ABB RobotStudio station: task2_Diaz_Raphael_20200421-193257.rsstn

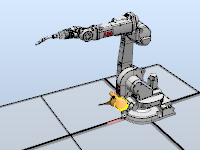
Station Solution2 (saved by RobotStudio 7.0.8732.594)
Controller IRB_1660ID_4kg_1.55m_1
  mechanical unit ROB_1: IRB1660ID_4_155__03, 6 joints, base frame (0, 0, 0) mm
Layout (positions relative to the parent item):
  - IRB1660ID_4_155__03 [mechanism, from Robots\IRB1660ID_4_155__03.rslib] at (0, 0, 0) mm; joint values [0, 0, 0, 0, 0, 0] (rad or m)
  - Binzel_ID_22 [mechanism, from Tools\Binzel_ID_22.rslib] at (962.96, 0, 1296.5) mm, rotated rx 0 ry 90 rz 0 deg
  - propeller [part, from Training Objects\propeller.rslib] at (600, 300, 492) mm
Attachment: Binzel_ID_22 is attached to IRB1660ID_4_155__03 / Link6
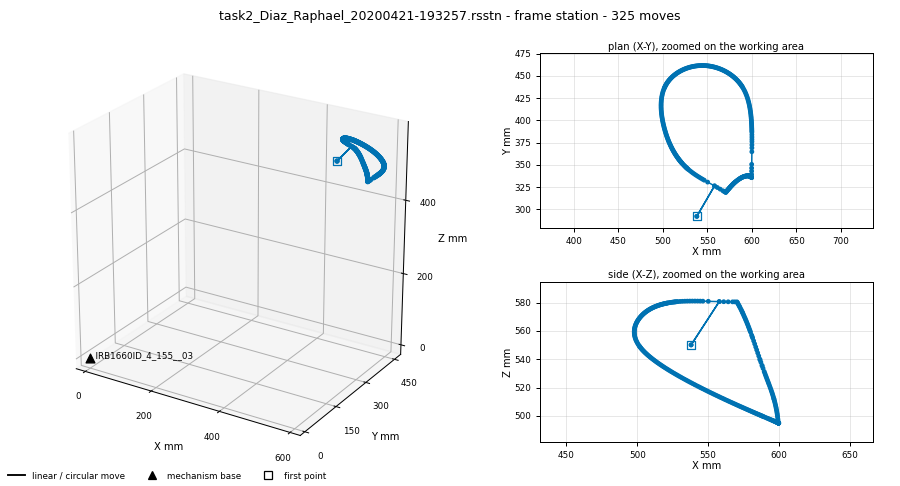
[picture p0: tool path of task2_Diaz_Raphael_20200421-193257.rsstn in frame station, 325 of 327 moves have a stored position in this frame; points joined in program order, loops and branches not executed]
Targets, tools, work objects and paths stored in the station, written as RAPID:
! task T_ROB1
MODULE CalibData
  PERS tooldata tWeldGun:=[TRUE,[[49.841566361,0,372.194826196],[0.981627183,0,0.190808995,0]],[2,[0,0,100],[0,1,0,0],0,0,0]];
  TASK PERS wobjdata wobjPropeller:=[FALSE,TRUE,"",[[600,300,492],[1,0,0,0]],[[0,0,0],[1,0,0,0]]];
ENDMODULE

! task T_ROB1
MODULE Module1
  CONST robtarget Target_10:=[[21.523963287,135.70517668,186.635026338],[0.089637387,-0.283764355,-0.851730307,0.431275333],[0,0,0,0],[9E+09,9E+09,9E+09,9E+09,9E+09,9E+09]];
  CONST robtarget Target_20:=[[-42.068819563,26.298976235,88.725674008],[0.089637387,-0.283764355,-0.851730307,0.431275333],[0,-1,-1,0],[9E+09,9E+09,9E+09,9E+09,9E+09,9E+09]];
  CONST robtarget Target_30:=[[-97.077163645,86.355573847,78.63839948],[0.089637387,-0.283764355,-0.851730307,0.431275333],[0,-1,-1,0],[9E+09,9E+09,9E+09,9E+09,9E+09,9E+09]];
  CONST robtarget Target_40:=[[-83.254485532,153.616685275,43.88735717],[0.089637387,-0.283764355,-0.851730307,0.431275333],[0,-1,-1,0],[9E+09,9E+09,9E+09,9E+09,9E+09,9E+09]];
  CONST robtarget Target_50:=[[-25.422721424,152.293184907,13.845629776],[0.089637387,-0.283764355,-0.851730307,0.431275333],[0,-1,-1,0],[9E+09,9E+09,9E+09,9E+09,9E+09,9E+09]];
  CONST robtarget Target_60:=[[-0.191127564,89.526890776,2.972180009],[0.089637387,-0.283764355,-0.851730307,0.431275333],[0,-1,-1,0],[9E+09,9E+09,9E+09,9E+09,9E+09,9E+09]];
  CONST robtarget Target_70:=[[-0.498093154,35.725710758,4.107130917],[0.089637387,-0.283764355,-0.851730307,0.431275333],[0,-1,-1,0],[9E+09,9E+09,9E+09,9E+09,9E+09,9E+09]];
  CONST robtarget Target_80:=[[-6.062970693,37.537743156,28.012491985],[0.089637387,-0.283764355,-0.851730307,0.431275333],[0,-1,-1,0],[9E+09,9E+09,9E+09,9E+09,9E+09,9E+09]];
  CONST robtarget Target_90:=[[-29.579108704,18.917792453,88.550574629],[0.089637387,-0.283764355,-0.851730307,0.431275333],[0,-1,-1,0],[9E+09,9E+09,9E+09,9E+09,9E+09,9E+09]];
  CONST robtarget Target_100:=[[-42.068819563,26.298976235,88.725674008],[0.089637387,-0.283764355,-0.851730307,0.431275333],[0,-1,-1,0],[9E+09,9E+09,9E+09,9E+09,9E+09,9E+09]];
  CONST robtarget Target_110:=[[-61.941679565,-7.890397172,58.129004558],[0.089637387,-0.283764355,-0.851730307,0.431275333],[0,-1,-1,0],[9E+09,9E+09,9E+09,9E+09,9E+09,9E+09]];
  CONST robtarget Target_120:=[[-61.941564206,-7.890461448,58.129001455],[0.089637387,-0.283764355,-0.851730307,0.431275333],[0,0,0,0],[9E+09,9E+09,9E+09,9E+09,9E+09,9E+09]];
  CONST robtarget Target_130:=[[-42.068819563,26.298976235,88.725674008],[0.089637387,-0.283764355,-0.851730307,0.431275333],[0,0,0,0],[9E+09,9E+09,9E+09,9E+09,9E+09,9E+09]];
  CONST robtarget Target_140:=[[-49.791866469,30.580230673,88.941782186],[0.089637387,-0.283764355,-0.851730307,0.431275333],[0,0,0,0],[9E+09,9E+09,9E+09,9E+09,9E+09,9E+09]];
  CONST robtarget Target_150:=[[-53.614959938,32.739613246,89.033496579],[0.089637387,-0.283764355,-0.851730307,0.431275333],[0,0,0,0],[9E+09,9E+09,9E+09,9E+09,9E+09,9E+09]];
  CONST robtarget Target_160:=[[-55.505547901,33.834166182,89.068675291],[0.089637387,-0.283764355,-0.851730307,0.431275333],[0,0,0,0],[9E+09,9E+09,9E+09,9E+09,9E+09,9E+09]];
  CONST robtarget Target_170:=[[-57.377839054,34.942502242,89.094223182],[0.089637387,-0.283764355,-0.851730307,0.431275333],[0,0,0,0],[9E+09,9E+09,9E+09,9E+09,9E+09,9E+09]];
  CONST robtarget Target_180:=[[-59.228590176,36.067527941,89.108256377],[0.089637387,-0.283764355,-0.851730307,0.431275333],[0,0,0,0],[9E+09,9E+09,9E+09,9E+09,9E+09,9E+09]];
  CONST robtarget Target_190:=[[-61.054558046,37.212149798,89.108891001],[0.089637387,-0.283764355,-0.851730307,0.431275333],[0,0,0,0],[9E+09,9E+09,9E+09,9E+09,9E+09,9E+09]];
  CONST robtarget Target_200:=[[-62.852499441,38.379274331,89.094243181],[0.089637387,-0.283764355,-0.851730307,0.431275333],[0,0,0,0],[9E+09,9E+09,9E+09,9E+09,9E+09,9E+09]];
  CONST robtarget Target_210:=[[-64.61917114,39.571808055,89.062429041],[0.089637387,-0.283764355,-0.851730307,0.431275333],[0,0,0,0],[9E+09,9E+09,9E+09,9E+09,9E+09,9E+09]];
  CONST robtarget Target_220:=[[-66.351329922,40.79265749,89.011564709],[0.089637387,-0.283764355,-0.851730307,0.431275333],[0,0,0,0],[9E+09,9E+09,9E+09,9E+09,9E+09,9E+09]];
  CONST robtarget Target_230:=[[-68.045732565,42.044729152,88.939766309],[0.089637387,-0.283764355,-0.851730307,0.431275333],[0,0,0,0],[9E+09,9E+09,9E+09,9E+09,9E+09,9E+09]];
  CONST robtarget Target_240:=[[-69.699135847,43.330929558,88.845149967],[0.089637387,-0.283764355,-0.851730307,0.431275333],[0,0,0,0],[9E+09,9E+09,9E+09,9E+09,9E+09,9E+09]];
  CONST robtarget Target_250:=[[-71.342075478,44.682787572,88.723134141],[0.089637387,-0.283764355,-0.851730307,0.431275333],[0,0,0,0],[9E+09,9E+09,9E+09,9E+09,9E+09,9E+09]];
  CONST robtarget Target_260:=[[-72.060749116,45.300688417,88.659667958],[0.089637387,-0.283764355,-0.851730307,0.431275333],[0,0,0,0],[9E+09,9E+09,9E+09,9E+09,9E+09,9E+09]];
  CONST robtarget Target_270:=[[-72.761042326,45.919421354,88.591393963],[0.089637387,-0.283764355,-0.851730307,0.431275333],[0,0,0,0],[9E+09,9E+09,9E+09,9E+09,9E+09,9E+09]];
  CONST robtarget Target_280:=[[-73.192658943,46.30937181,88.54602645],[0.089637387,-0.283764355,-0.851730307,0.431275333],[0,0,0,0],[9E+09,9E+09,9E+09,9E+09,9E+09,9E+09]];
  CONST robtarget Target_290:=[[-73.676857993,46.754481273,88.492204842],[0.089637387,-0.283764355,-0.851730307,0.431275333],[0,0,0,0],[9E+09,9E+09,9E+09,9E+09,9E+09,9E+09]];
  CONST robtarget Target_300:=[[-74.211820015,47.256226874,88.428916141],[0.089637387,-0.283764355,-0.851730307,0.431275333],[0,0,0,0],[9E+09,9E+09,9E+09,9E+09,9E+09,9E+09]];
  CONST robtarget Target_310:=[[-74.795612514,47.816163555,88.355085942],[0.089637387,-0.283764355,-0.851730307,0.431275333],[0,0,0,0],[9E+09,9E+09,9E+09,9E+09,9E+09,9E+09]];
  CONST robtarget Target_320:=[[-75.426303,48.435846257,88.269639843],[0.089637387,-0.283764355,-0.851730307,0.431275333],[0,0,0,0],[9E+09,9E+09,9E+09,9E+09,9E+09,9E+09]];
  CONST robtarget Target_330:=[[-76.101837442,49.116922118,88.171436479],[0.089637387,-0.283764355,-0.851730307,0.431275333],[0,0,0,0],[9E+09,9E+09,9E+09,9E+09,9E+09,9E+09]];
  CONST robtarget Target_340:=[[-76.819730038,49.861315108,88.059102158],[0.089637387,-0.283764355,-0.851730307,0.431275333],[0,0,0,0],[9E+09,9E+09,9E+09,9E+09,9E+09,9E+09]];
  CONST robtarget Target_350:=[[-77.577400632,50.670995418,87.931213982],[0.089637387,-0.283764355,-0.851730307,0.431275333],[0,0,0,0],[9E+09,9E+09,9E+09,9E+09,9E+09,9E+09]];
  CONST robtarget Target_360:=[[-78.37226907,51.547933238,87.786349051],[0.089637387,-0.283764355,-0.851730307,0.431275333],[0,0,0,0],[9E+09,9E+09,9E+09,9E+09,9E+09,9E+09]];
  CONST robtarget Target_370:=[[-78.78283064,52.012251515,87.70709705],[0.089637387,-0.283764355,-0.851730307,0.431275333],[0,0,0,0],[9E+09,9E+09,9E+09,9E+09,9E+09,9E+09]];
  CONST robtarget Target_380:=[[-79.201648961,52.494165078,87.623027502],[0.089637387,-0.283764355,-0.851730307,0.431275333],[0,0,0,0],[9E+09,9E+09,9E+09,9E+09,9E+09,9E+09]];
  CONST robtarget Target_390:=[[-79.628335409,52.993946989,87.533928686],[0.089637387,-0.283764355,-0.851730307,0.431275333],[0,0,0,0],[9E+09,9E+09,9E+09,9E+09,9E+09,9E+09]];
  CONST robtarget Target_400:=[[-80.062501358,53.511870309,87.439588878],[0.089637387,-0.283764355,-0.851730307,0.431275333],[0,0,0,0],[9E+09,9E+09,9E+09,9E+09,9E+09,9E+09]];
  CONST robtarget Target_410:=[[-80.503758184,54.048208097,87.339796355],[0.089637387,-0.283764355,-0.851730307,0.431275333],[0,0,0,0],[9E+09,9E+09,9E+09,9E+09,9E+09,9E+09]];
  CONST robtarget Target_420:=[[-80.951717264,54.603233414,87.234339393],[0.089637387,-0.283764355,-0.851730307,0.431275333],[0,0,0,0],[9E+09,9E+09,9E+09,9E+09,9E+09,9E+09]];
  CONST robtarget Target_430:=[[-81.405989972,55.177219322,87.123006269],[0.089637387,-0.283764355,-0.851730307,0.431275333],[0,0,0,0],[9E+09,9E+09,9E+09,9E+09,9E+09,9E+09]];
  CONST robtarget Target_440:=[[-81.866187684,55.77043888,87.005585259],[0.089637387,-0.283764355,-0.851730307,0.431275333],[0,0,0,0],[9E+09,9E+09,9E+09,9E+09,9E+09,9E+09]];
  CONST robtarget Target_450:=[[-82.331908288,56.383173791,86.881857385],[0.089637387,-0.283764355,-0.851730307,0.431275333],[0,0,0,0],[9E+09,9E+09,9E+09,9E+09,9E+09,9E+09]];
  CONST robtarget Target_460:=[[-82.802718317,57.015702111,86.751589396],[0.089637387,-0.283764355,-0.851730307,0.431275333],[0,0,0,0],[9E+09,9E+09,9E+09,9E+09,9E+09,9E+09]];
  CONST robtarget Target_470:=[[-83.278182117,57.668291429,86.614548166],[0.089637387,-0.283764355,-0.851730307,0.431275333],[0,0,0,0],[9E+09,9E+09,9E+09,9E+09,9E+09,9E+09]];
  CONST robtarget Target_480:=[[-83.75786403,58.341209334,86.470500568],[0.089637387,-0.283764355,-0.851730307,0.431275333],[0,0,0,0],[9E+09,9E+09,9E+09,9E+09,9E+09,9E+09]];
  CONST robtarget Target_490:=[[-84.2413284,59.034723416,86.319213476],[0.089637387,-0.283764355,-0.851730307,0.431275333],[0,0,0,0],[9E+09,9E+09,9E+09,9E+09,9E+09,9E+09]];
  CONST robtarget Target_500:=[[-84.728139572,59.749101264,86.160453763],[0.089637387,-0.283764355,-0.851730307,0.431275333],[0,0,0,0],[9E+09,9E+09,9E+09,9E+09,9E+09,9E+09]];
  CONST robtarget Target_510:=[[-85.21786189,60.484610466,85.993988302],[0.089637387,-0.283764355,-0.851730307,0.431275333],[0,0,0,0],[9E+09,9E+09,9E+09,9E+09,9E+09,9E+09]];
  CONST robtarget Target_520:=[[-85.710059697,61.241518614,85.819583966],[0.089637387,-0.283764355,-0.851730307,0.431275333],[0,0,0,0],[9E+09,9E+09,9E+09,9E+09,9E+09,9E+09]];
  CONST robtarget Target_530:=[[-86.204286606,62.020097275,85.637002174],[0.089637387,-0.283764355,-0.851730307,0.431275333],[0,0,0,0],[9E+09,9E+09,9E+09,9E+09,9E+09,9E+09]];
  CONST robtarget Target_540:=[[-86.700080407,62.820588107,85.446000215],[0.089637387,-0.283764355,-0.851730307,0.431275333],[0,0,0,0],[9E+09,9E+09,9E+09,9E+09,9E+09,9E+09]];
  CONST robtarget Target_550:=[[-87.196981704,63.643213831,85.246338775],[0.089637387,-0.283764355,-0.851730307,0.431275333],[0,0,0,0],[9E+09,9E+09,9E+09,9E+09,9E+09,9E+09]];
  CONST robtarget Target_560:=[[-87.694531106,64.488197169,85.037778537],[0.089637387,-0.283764355,-0.851730307,0.431275333],[0,0,0,0],[9E+09,9E+09,9E+09,9E+09,9E+09,9E+09]];
  CONST robtarget Target_570:=[[-88.192269217,65.355760842,84.820080186],[0.089637387,-0.283764355,-0.851730307,0.431275333],[0,0,0,0],[9E+09,9E+09,9E+09,9E+09,9E+09,9E+09]];
  CONST robtarget Target_580:=[[-88.689736644,66.246127572,84.593004406],[0.089637387,-0.283764355,-0.851730307,0.431275333],[0,0,0,0],[9E+09,9E+09,9E+09,9E+09,9E+09,9E+09]];
  CONST robtarget Target_590:=[[-89.186473995,67.159520081,84.356311882],[0.089637387,-0.283764355,-0.851730307,0.431275333],[0,0,0,0],[9E+09,9E+09,9E+09,9E+09,9E+09,9E+09]];
  CONST robtarget Target_600:=[[-89.682021875,68.09616109,84.109763297],[0.089637387,-0.283764355,-0.851730307,0.431275333],[0,0,0,0],[9E+09,9E+09,9E+09,9E+09,9E+09,9E+09]];
  CONST robtarget Target_610:=[[-90.175913619,69.056271448,83.853116141],[0.089637387,-0.283764355,-0.851730307,0.431275333],[0,0,0,0],[9E+09,9E+09,9E+09,9E+09,9E+09,9E+09]];
  CONST robtarget Target_620:=[[-90.667685083,70.040011068,83.586135756],[0.089637387,-0.283764355,-0.851730307,0.431275333],[0,0,0,0],[9E+09,9E+09,9E+09,9E+09,9E+09,9E+09]];
  CONST robtarget Target_630:=[[-91.15688065,71.04751127,83.308594608],[0.089637387,-0.283764355,-0.851730307,0.431275333],[0,0,0,0],[9E+09,9E+09,9E+09,9E+09,9E+09,9E+09]];
  CONST robtarget Target_640:=[[-91.643044702,72.078903372,83.020265165],[0.089637387,-0.283764355,-0.851730307,0.431275333],[0,0,0,0],[9E+09,9E+09,9E+09,9E+09,9E+09,9E+09]];
  CONST robtarget Target_650:=[[-92.125721625,73.134318692,82.720919892],[0.089637387,-0.283764355,-0.851730307,0.431275333],[0,0,0,0],[9E+09,9E+09,9E+09,9E+09,9E+09,9E+09]];
  CONST robtarget Target_660:=[[-92.604455801,74.21388855,82.410331256],[0.089637387,-0.283764355,-0.851730307,0.431275333],[0,0,0,0],[9E+09,9E+09,9E+09,9E+09,9E+09,9E+09]];
  CONST robtarget Target_670:=[[-93.078791613,75.317744264,82.088271723],[0.089637387,-0.283764355,-0.851730307,0.431275333],[0,0,0,0],[9E+09,9E+09,9E+09,9E+09,9E+09,9E+09]];
  CONST robtarget Target_680:=[[-93.548273446,76.446017152,81.754513761],[0.089637387,-0.283764355,-0.851730307,0.431275333],[0,0,0,0],[9E+09,9E+09,9E+09,9E+09,9E+09,9E+09]];
  CONST robtarget Target_690:=[[-94.012442576,77.598829619,81.408829359],[0.089637387,-0.283764355,-0.851730307,0.431275333],[0,0,0,0],[9E+09,9E+09,9E+09,9E+09,9E+09,9E+09]];
  CONST robtarget Target_700:=[[-94.470863955,78.776207351,81.051012179],[0.089637387,-0.283764355,-0.851730307,0.431275333],[0,0,0,0],[9E+09,9E+09,9E+09,9E+09,9E+09,9E+09]];
  CONST robtarget Target_710:=[[-94.92311748,79.978136589,80.6808672],[0.089637387,-0.283764355,-0.851730307,0.431275333],[0,0,0,0],[9E+09,9E+09,9E+09,9E+09,9E+09,9E+09]];
  CONST robtarget Target_720:=[[-95.368783045,81.204603576,80.298199397],[0.089637387,-0.283764355,-0.851730307,0.431275333],[0,0,0,0],[9E+09,9E+09,9E+09,9E+09,9E+09,9E+09]];
  CONST robtarget Target_730:=[[-95.807440548,82.455594554,79.902813746],[0.089637387,-0.283764355,-0.851730307,0.431275333],[0,0,0,0],[9E+09,9E+09,9E+09,9E+09,9E+09,9E+09]];
  CONST robtarget Target_740:=[[-96.238669885,83.731095764,79.494515226],[0.089637387,-0.283764355,-0.851730307,0.431275333],[0,0,0,0],[9E+09,9E+09,9E+09,9E+09,9E+09,9E+09]];
  CONST robtarget Target_750:=[[-96.662050952,85.031093447,79.073108811],[0.089637387,-0.283764355,-0.851730307,0.431275333],[0,0,0,0],[9E+09,9E+09,9E+09,9E+09,9E+09,9E+09]];
  CONST robtarget Target_760:=[[-97.077163645,86.355573847,78.63839948],[0.089637387,-0.283764355,-0.851730307,0.431275333],[0,0,0,0],[9E+09,9E+09,9E+09,9E+09,9E+09,9E+09]];
  CONST robtarget Target_770:=[[-97.483682077,87.704485468,78.19021474],[0.089637387,-0.283764355,-0.851730307,0.431275333],[0,0,0,0],[9E+09,9E+09,9E+09,9E+09,9E+09,9E+09]];
  CONST robtarget Target_780:=[[-97.881197354,89.077633701,77.728399267],[0.089637387,-0.283764355,-0.851730307,0.431275333],[0,0,0,0],[9E+09,9E+09,9E+09,9E+09,9E+09,9E+09]];
  CONST robtarget Target_790:=[[-98.269164855,90.47479012,77.252783791],[0.089637387,-0.283764355,-0.851730307,0.431275333],[0,0,0,0],[9E+09,9E+09,9E+09,9E+09,9E+09,9E+09]];
  CONST robtarget Target_800:=[[-98.647039962,91.895726298,76.763199041],[0.089637387,-0.283764355,-0.851730307,0.431275333],[0,0,0,0],[9E+09,9E+09,9E+09,9E+09,9E+09,9E+09]];
  CONST robtarget Target_810:=[[-99.013905738,93.340048971,76.259451373],[0.089637387,-0.283764355,-0.851730307,0.431275333],[0,0,0,0],[9E+09,9E+09,9E+09,9E+09,9E+09,9E+09]];
  CONST robtarget Target_820:=[[-99.368243888,94.807039694,75.741321273],[0.089637387,-0.283764355,-0.851730307,0.431275333],[0,0,0,0],[9E+09,9E+09,9E+09,9E+09,9E+09,9E+09]];
  CONST robtarget Target_830:=[[-99.708607753,96.295982268,75.208600662],[0.089637387,-0.283764355,-0.851730307,0.431275333],[0,0,0,0],[9E+09,9E+09,9E+09,9E+09,9E+09,9E+09]];
  CONST robtarget Target_840:=[[-100.033550677,97.806160497,74.661081462],[0.089637387,-0.283764355,-0.851730307,0.431275333],[0,0,0,0],[9E+09,9E+09,9E+09,9E+09,9E+09,9E+09]];
  CONST robtarget Target_850:=[[-100.341583594,99.336818217,74.098557633],[0.089637387,-0.283764355,-0.851730307,0.431275333],[0,0,0,0],[9E+09,9E+09,9E+09,9E+09,9E+09,9E+09]];
  CONST robtarget Target_860:=[[-100.631031883,100.8870215,73.520833315],[0.089637387,-0.283764355,-0.851730307,0.431275333],[0,0,0,0],[9E+09,9E+09,9E+09,9E+09,9E+09,9E+09]];
  CONST robtarget Target_870:=[[-100.900170557,102.455787493,72.927715696],[0.089637387,-0.283764355,-0.851730307,0.431275333],[0,0,0,0],[9E+09,9E+09,9E+09,9E+09,9E+09,9E+09]];
  CONST robtarget Target_880:=[[-101.147274629,104.042133343,72.319011966],[0.089637387,-0.283764355,-0.851730307,0.431275333],[0,0,0,0],[9E+09,9E+09,9E+09,9E+09,9E+09,9E+09]];
  CONST robtarget Target_890:=[[-101.370571802,105.645030719,71.694531974],[0.089637387,-0.283764355,-0.851730307,0.431275333],[0,0,0,0],[9E+09,9E+09,9E+09,9E+09,9E+09,9E+09]];
  CONST robtarget Target_900:=[[-101.568083835,107.263250566,71.054098336],[0.089637387,-0.283764355,-0.851730307,0.431275333],[0,0,0,0],[9E+09,9E+09,9E+09,9E+09,9E+09,9E+09]];
  CONST robtarget Target_910:=[[-101.737776824,108.895508939,70.397537389],[0.089637387,-0.283764355,-0.851730307,0.431275333],[0,0,0,0],[9E+09,9E+09,9E+09,9E+09,9E+09,9E+09]];
  CONST robtarget Target_920:=[[-101.877616866,110.540521898,69.724675469],[0.089637387,-0.283764355,-0.851730307,0.431275333],[0,0,0,0],[9E+09,9E+09,9E+09,9E+09,9E+09,9E+09]];
  CONST robtarget Target_930:=[[-101.985517598,112.196954226,69.035342228],[0.089637387,-0.283764355,-0.851730307,0.431275333],[0,0,0,0],[9E+09,9E+09,9E+09,9E+09,9E+09,9E+09]];
  CONST robtarget Target_940:=[[-102.059165334,113.863245906,68.329382794],[0.089637387,-0.283764355,-0.851730307,0.431275333],[0,0,0,0],[9E+09,9E+09,9E+09,9E+09,9E+09,9E+09]];
  CONST robtarget Target_950:=[[-102.096185174,115.537775795,67.606646723],[0.089637387,-0.283764355,-0.851730307,0.431275333],[0,0,0,0],[9E+09,9E+09,9E+09,9E+09,9E+09,9E+09]];
  CONST robtarget Target_960:=[[-102.094202223,117.218922746,66.866983568],[0.089637387,-0.283764355,-0.851730307,0.431275333],[0,0,0,0],[9E+09,9E+09,9E+09,9E+09,9E+09,9E+09]];
  CONST robtarget Target_970:=[[-102.050783732,118.905008267,66.110246882],[0.089637387,-0.283764355,-0.851730307,0.431275333],[0,0,0,0],[9E+09,9E+09,9E+09,9E+09,9E+09,9E+09]];
  CONST robtarget Target_980:=[[-101.963247246,120.594103871,65.336308536],[0.089637387,-0.283764355,-0.851730307,0.431275333],[0,0,0,0],[9E+09,9E+09,9E+09,9E+09,9E+09,9E+09]];
  CONST robtarget Target_990:=[[-101.82884331,122.284213421,64.545045559],[0.089637387,-0.283764355,-0.851730307,0.431275333],[0,0,0,0],[9E+09,9E+09,9E+09,9E+09,9E+09,9E+09]];
  CONST robtarget Target_1000:=[[-101.644822469,123.973340779,63.736334981],[0.089637387,-0.283764355,-0.851730307,0.431275333],[0,0,0,0],[9E+09,9E+09,9E+09,9E+09,9E+09,9E+09]];
  CONST robtarget Target_1010:=[[-101.408371772,125.659426107,62.910058546],[0.089637387,-0.283764355,-0.851730307,0.431275333],[0,0,0,0],[9E+09,9E+09,9E+09,9E+09,9E+09,9E+09]];
  CONST robtarget Target_1020:=[[-101.116405192,127.340133258,62.066119282],[0.089637387,-0.283764355,-0.851730307,0.431275333],[0,0,0,0],[9E+09,9E+09,9E+09,9E+09,9E+09,9E+09]];
  CONST robtarget Target_1030:=[[-100.765763661,129.013051638,61.204426141],[0.089637387,-0.283764355,-0.851730307,0.431275333],[0,0,0,0],[9E+09,9E+09,9E+09,9E+09,9E+09,9E+09]];
  CONST robtarget Target_1040:=[[-100.353288111,130.675770651,60.324888075],[0.089637387,-0.283764355,-0.851730307,0.431275333],[0,0,0,0],[9E+09,9E+09,9E+09,9E+09,9E+09,9E+09]];
  CONST robtarget Target_1050:=[[-99.875750085,132.325809364,59.4274195],[0.089637387,-0.283764355,-0.851730307,0.431275333],[0,0,0,0],[9E+09,9E+09,9E+09,9E+09,9E+09,9E+09]];
  CONST robtarget Target_1060:=[[-99.329623689,133.96038311,58.511959204],[0.089637387,-0.283764355,-0.851730307,0.431275333],[0,0,0,0],[9E+09,9E+09,9E+09,9E+09,9E+09,9E+09]];
  CONST robtarget Target_1070:=[[-98.711303696,135.57662569,57.578452699],[0.089637387,-0.283764355,-0.851730307,0.431275333],[0,0,0,0],[9E+09,9E+09,9E+09,9E+09,9E+09,9E+09]];
  CONST robtarget Target_1080:=[[-98.373944468,136.376977106,57.10491509],[0.089637387,-0.283764355,-0.851730307,0.431275333],[0,0,0,0],[9E+09,9E+09,9E+09,9E+09,9E+09,9E+09]];
  CONST robtarget Target_1090:=[[-98.01718488,137.171670907,56.626845496],[0.089637387,-0.283764355,-0.851730307,0.431275333],[0,0,0,0],[9E+09,9E+09,9E+09,9E+09,9E+09,9E+09]];
  CONST robtarget Target_1100:=[[-97.640535504,137.960322993,56.144237301],[0.089637387,-0.283764355,-0.851730307,0.431275333],[0,0,0,0],[9E+09,9E+09,9E+09,9E+09,9E+09,9E+09]];
  CONST robtarget Target_1110:=[[-97.243501368,138.742523396,55.657088796],[0.089637387,-0.283764355,-0.851730307,0.431275333],[0,0,0,0],[9E+09,9E+09,9E+09,9E+09,9E+09,9E+09]];
  CONST robtarget Target_1120:=[[-96.825623509,139.517875036,55.165400527],[0.089637387,-0.283764355,-0.851730307,0.431275333],[0,0,0,0],[9E+09,9E+09,9E+09,9E+09,9E+09,9E+09]];
  CONST robtarget Target_1130:=[[-96.386442962,140.28598083,54.669173042],[0.089637387,-0.283764355,-0.851730307,0.431275333],[0,0,0,0],[9E+09,9E+09,9E+09,9E+09,9E+09,9E+09]];
  CONST robtarget Target_1140:=[[-95.925711374,141.046481587,54.168428273],[0.089637387,-0.283764355,-0.851730307,0.431275333],[0,0,0,0],[9E+09,9E+09,9E+09,9E+09,9E+09,9E+09]];
  CONST robtarget Target_1150:=[[-95.443552762,141.799075074,53.663228181],[0.089637387,-0.283764355,-0.851730307,0.431275333],[0,0,0,0],[9E+09,9E+09,9E+09,9E+09,9E+09,9E+09]];
  CONST robtarget Target_1160:=[[-94.940066713,142.543449653,53.153633355],[0.089637387,-0.283764355,-0.851730307,0.431275333],[0,0,0,0],[9E+09,9E+09,9E+09,9E+09,9E+09,9E+09]];
  CONST robtarget Target_1170:=[[-94.415352815,143.279293685,52.639704389],[0.089637387,-0.283764355,-0.851730307,0.431275333],[0,0,0,0],[9E+09,9E+09,9E+09,9E+09,9E+09,9E+09]];
  CONST robtarget Target_1180:=[[-93.869500391,144.006300939,52.121499208],[0.089637387,-0.283764355,-0.851730307,0.431275333],[0,0,0,0],[9E+09,9E+09,9E+09,9E+09,9E+09,9E+09]];
  CONST robtarget Target_1190:=[[-93.302636325,144.724144959,51.59908555],[0.089637387,-0.283764355,-0.851730307,0.431275333],[0,0,0,0],[9E+09,9E+09,9E+09,9E+09,9E+09,9E+09]];
  CONST robtarget Target_1200:=[[-92.71491655,145.432483766,51.072538723],[0.089637387,-0.283764355,-0.851730307,0.431275333],[0,0,0,0],[9E+09,9E+09,9E+09,9E+09,9E+09,9E+09]];
  CONST robtarget Target_1210:=[[-92.106496997,146.13097538,50.541934035],[0.089637387,-0.283764355,-0.851730307,0.431275333],[0,0,0,0],[9E+09,9E+09,9E+09,9E+09,9E+09,9E+09]];
  CONST robtarget Target_1220:=[[-91.477533598,146.819277823,50.007346793],[0.089637387,-0.283764355,-0.851730307,0.431275333],[0,0,0,0],[9E+09,9E+09,9E+09,9E+09,9E+09,9E+09]];
  CONST robtarget Target_1230:=[[-90.828182284,147.497049114,49.468852306],[0.089637387,-0.283764355,-0.851730307,0.431275333],[0,0,0,0],[9E+09,9E+09,9E+09,9E+09,9E+09,9E+09]];
  CONST robtarget Target_1240:=[[-90.158598987,148.163947276,48.926525883],[0.089637387,-0.283764355,-0.851730307,0.431275333],[0,0,0,0],[9E+09,9E+09,9E+09,9E+09,9E+09,9E+09]];
  CONST robtarget Target_1250:=[[-89.468939638,148.819630327,48.38044283],[0.089637387,-0.283764355,-0.851730307,0.431275333],[0,0,0,0],[9E+09,9E+09,9E+09,9E+09,9E+09,9E+09]];
  CONST robtarget Target_1260:=[[-88.759371673,149.463749958,47.83068148],[0.089637387,-0.283764355,-0.851730307,0.431275333],[0,0,0,0],[9E+09,9E+09,9E+09,9E+09,9E+09,9E+09]];
  CONST robtarget Target_1270:=[[-88.030117086,150.095929082,47.277334333],[0.089637387,-0.283764355,-0.851730307,0.431275333],[0,0,0,0],[9E+09,9E+09,9E+09,9E+09,9E+09,9E+09]];
  CONST robtarget Target_1280:=[[-87.281413645,150.715782558,46.72049795],[0.089637387,-0.283764355,-0.851730307,0.431275333],[0,0,0,0],[9E+09,9E+09,9E+09,9E+09,9E+09,9E+09]];
  CONST robtarget Target_1290:=[[-86.513499118,151.322925246,46.160268893],[0.089637387,-0.283764355,-0.851730307,0.431275333],[0,0,0,0],[9E+09,9E+09,9E+09,9E+09,9E+09,9E+09]];
  CONST robtarget Target_1300:=[[-85.726611275,151.916972002,45.596743725],[0.089637387,-0.283764355,-0.851730307,0.431275333],[0,0,0,0],[9E+09,9E+09,9E+09,9E+09,9E+09,9E+09]];
  CONST robtarget Target_1310:=[[-84.920987884,152.497537687,45.030019008],[0.089637387,-0.283764355,-0.851730307,0.431275333],[0,0,0,0],[9E+09,9E+09,9E+09,9E+09,9E+09,9E+09]];
  CONST robtarget Target_1320:=[[-84.096866713,153.064237158,44.460191302],[0.089637387,-0.283764355,-0.851730307,0.431275333],[0,0,0,0],[9E+09,9E+09,9E+09,9E+09,9E+09,9E+09]];
  CONST robtarget Target_1330:=[[-83.254485532,153.616685275,43.88735717],[0.089637387,-0.283764355,-0.851730307,0.431275333],[0,0,0,0],[9E+09,9E+09,9E+09,9E+09,9E+09,9E+09]];
  CONST robtarget Target_1340:=[[-82.394094894,154.154490046,43.311616509],[0.089637387,-0.283764355,-0.851730307,0.431275333],[0,0,0,0],[9E+09,9E+09,9E+09,9E+09,9E+09,9E+09]];
  CONST robtarget Target_1350:=[[-81.516005347,154.677228513,42.733084706],[0.089637387,-0.283764355,-0.851730307,0.431275333],[0,0,0,0],[9E+09,9E+09,9E+09,9E+09,9E+09,9E+09]];
  CONST robtarget Target_1360:=[[-80.620544648,155.184469083,42.151881558],[0.089637387,-0.283764355,-0.851730307,0.431275333],[0,0,0,0],[9E+09,9E+09,9E+09,9E+09,9E+09,9E+09]];
  CONST robtarget Target_1370:=[[-79.708040553,155.675780162,41.568126862],[0.089637387,-0.283764355,-0.851730307,0.431275333],[0,0,0,0],[9E+09,9E+09,9E+09,9E+09,9E+09,9E+09]];
  CONST robtarget Target_1380:=[[-78.778820818,156.150730158,40.981940416],[0.089637387,-0.283764355,-0.851730307,0.431275333],[0,0,0,0],[9E+09,9E+09,9E+09,9E+09,9E+09,9E+09]];
  CONST robtarget Target_1390:=[[-77.833213201,156.608887477,40.393442017],[0.089637387,-0.283764355,-0.851730307,0.431275333],[0,0,0,0],[9E+09,9E+09,9E+09,9E+09,9E+09,9E+09]];
  CONST robtarget Target_1400:=[[-76.871545457,157.049820527,39.802751462],[0.089637387,-0.283764355,-0.851730307,0.431275333],[0,0,0,0],[9E+09,9E+09,9E+09,9E+09,9E+09,9E+09]];
  CONST robtarget Target_1410:=[[-75.894145343,157.473097712,39.209988548],[0.089637387,-0.283764355,-0.851730307,0.431275333],[0,0,0,0],[9E+09,9E+09,9E+09,9E+09,9E+09,9E+09]];
  CONST robtarget Target_1420:=[[-74.901354733,157.878280056,38.615276732],[0.089637387,-0.283764355,-0.851730307,0.431275333],[0,0,0,0],[9E+09,9E+09,9E+09,9E+09,9E+09,9E+09]];
  CONST robtarget Target_1430:=[[-73.893581114,158.264895339,38.018756325],[0.089637387,-0.283764355,-0.851730307,0.431275333],[0,0,0,0],[9E+09,9E+09,9E+09,9E+09,9E+09,9E+09]];
  CONST robtarget Target_1440:=[[-72.87125067,158.632462113,37.420572413],[0.089637387,-0.283764355,-0.851730307,0.431275333],[0,0,0,0],[9E+09,9E+09,9E+09,9E+09,9E+09,9E+09]];
  CONST robtarget Target_1450:=[[-71.834789579,158.980498927,36.820870078],[0.089637387,-0.283764355,-0.851730307,0.431275333],[0,0,0,0],[9E+09,9E+09,9E+09,9E+09,9E+09,9E+09]];
  CONST robtarget Target_1460:=[[-70.784624025,159.308524331,36.219794405],[0.089637387,-0.283764355,-0.851730307,0.431275333],[0,0,0,0],[9E+09,9E+09,9E+09,9E+09,9E+09,9E+09]];
  CONST robtarget Target_1470:=[[-69.721180188,159.616056875,35.617490477],[0.089637387,-0.283764355,-0.851730307,0.431275333],[0,0,0,0],[9E+09,9E+09,9E+09,9E+09,9E+09,9E+09]];
  CONST robtarget Target_1480:=[[-68.644884249,159.902615109,35.014103378],[0.089637387,-0.283764355,-0.851730307,0.431275333],[0,0,0,0],[9E+09,9E+09,9E+09,9E+09,9E+09,9E+09]];
  CONST robtarget Target_1490:=[[-67.55616239,160.167717582,34.409778192],[0.089637387,-0.283764355,-0.851730307,0.431275333],[0,0,0,0],[9E+09,9E+09,9E+09,9E+09,9E+09,9E+09]];
  CONST robtarget Target_1500:=[[-66.455479479,160.410863431,33.804669917],[0.089637387,-0.283764355,-0.851730307,0.431275333],[0,0,0,0],[9E+09,9E+09,9E+09,9E+09,9E+09,9E+09]];
  CONST robtarget Target_1510:=[[-65.343353291,160.631525372,33.198947094],[0.089637387,-0.283764355,-0.851730307,0.431275333],[0,0,0,0],[9E+09,9E+09,9E+09,9E+09,9E+09,9E+09]];
  CONST robtarget Target_1520:=[[-64.220289368,160.829182326,32.592775118],[0.089637387,-0.283764355,-0.851730307,0.431275333],[0,0,0,0],[9E+09,9E+09,9E+09,9E+09,9E+09,9E+09]];
  CONST robtarget Target_1530:=[[-63.086793249,161.003313214,31.986319384],[0.089637387,-0.283764355,-0.851730307,0.431275333],[0,0,0,0],[9E+09,9E+09,9E+09,9E+09,9E+09,9E+09]];
  CONST robtarget Target_1540:=[[-61.943384215,161.153390145,31.379748799],[0.089637387,-0.283764355,-0.851730307,0.431275333],[0,0,0,0],[9E+09,9E+09,9E+09,9E+09,9E+09,9E+09]];
  CONST robtarget Target_1550:=[[-60.790609276,161.278871503,30.77323935],[0.089637387,-0.283764355,-0.851730307,0.431275333],[0,0,0,0],[9E+09,9E+09,9E+09,9E+09,9E+09,9E+09]];
  CONST robtarget Target_1560:=[[-59.629020895,161.379212994,30.166968412],[0.089637387,-0.283764355,-0.851730307,0.431275333],[0,0,0,0],[9E+09,9E+09,9E+09,9E+09,9E+09,9E+09]];
  CONST robtarget Target_1570:=[[-58.605848224,161.44595514,29.636819659],[0.089637387,-0.283764355,-0.851730307,0.431275333],[0,0,0,0],[9E+09,9E+09,9E+09,9E+09,9E+09,9E+09]];
  CONST robtarget Target_1580:=[[-57.318566058,161.500963653,28.974738132],[0.089637387,-0.283764355,-0.851730307,0.431275333],[0,0,0,0],[9E+09,9E+09,9E+09,9E+09,9E+09,9E+09]];
  CONST robtarget Target_1590:=[[-56.179983218,161.522654054,28.393499156],[0.089637387,-0.283764355,-0.851730307,0.431275333],[0,0,0,0],[9E+09,9E+09,9E+09,9E+09,9E+09,9E+09]];
  CONST robtarget Target_1600:=[[-55.043993927,161.519276456,27.817513287],[0.089637387,-0.283764355,-0.851730307,0.431275333],[0,0,0,0],[9E+09,9E+09,9E+09,9E+09,9E+09,9E+09]];
  CONST robtarget Target_1610:=[[-53.911152598,161.491173917,27.246893168],[0.089637387,-0.283764355,-0.851730307,0.431275333],[0,0,0,0],[9E+09,9E+09,9E+09,9E+09,9E+09,9E+09]];
  CONST robtarget Target_1620:=[[-52.782013645,161.438689493,26.681751443],[0.089637387,-0.283764355,-0.851730307,0.431275333],[0,0,0,0],[9E+09,9E+09,9E+09,9E+09,9E+09,9E+09]];
  CONST robtarget Target_1630:=[[-51.657131483,161.362166244,26.122200755],[0.089637387,-0.283764355,-0.851730307,0.431275333],[0,0,0,0],[9E+09,9E+09,9E+09,9E+09,9E+09,9E+09]];
  CONST robtarget Target_1640:=[[-50.537060524,161.261947226,25.568353747],[0.089637387,-0.283764355,-0.851730307,0.431275333],[0,0,0,0],[9E+09,9E+09,9E+09,9E+09,9E+09,9E+09]];
  CONST robtarget Target_1650:=[[-49.422355184,161.138375497,25.020323063],[0.089637387,-0.283764355,-0.851730307,0.431275333],[0,0,0,0],[9E+09,9E+09,9E+09,9E+09,9E+09,9E+09]];
  CONST robtarget Target_1660:=[[-48.31354999,160.991943178,24.478225714],[0.089637387,-0.283764355,-0.851730307,0.431275333],[0,0,0,0],[9E+09,9E+09,9E+09,9E+09,9E+09,9E+09]];
  CONST robtarget Target_1670:=[[-47.211113798,160.82319606,23.942165647],[0.089637387,-0.283764355,-0.851730307,0.431275333],[0,0,0,0],[9E+09,9E+09,9E+09,9E+09,9E+09,9E+09]];
  CONST robtarget Target_1680:=[[-46.115502514,160.632557701,23.412235913],[0.089637387,-0.283764355,-0.851730307,0.431275333],[0,0,0,0],[9E+09,9E+09,9E+09,9E+09,9E+09,9E+09]];
  CONST robtarget Target_1690:=[[-45.027172042,160.42045166,22.888529564],[0.089637387,-0.283764355,-0.851730307,0.431275333],[0,0,0,0],[9E+09,9E+09,9E+09,9E+09,9E+09,9E+09]];
  CONST robtarget Target_1700:=[[-43.946578289,160.187301498,22.371139651],[0.089637387,-0.283764355,-0.851730307,0.431275333],[0,0,0,0],[9E+09,9E+09,9E+09,9E+09,9E+09,9E+09]];
  CONST robtarget Target_1710:=[[-42.87417716,159.933530773,21.860159223],[0.089637387,-0.283764355,-0.851730307,0.431275333],[0,0,0,0],[9E+09,9E+09,9E+09,9E+09,9E+09,9E+09]];
  CONST robtarget Target_1720:=[[-41.810424561,159.659563045,21.355681333],[0.089637387,-0.283764355,-0.851730307,0.431275333],[0,0,0,0],[9E+09,9E+09,9E+09,9E+09,9E+09,9E+09]];
  CONST robtarget Target_1730:=[[-40.755776397,159.365821874,20.857799032],[0.089637387,-0.283764355,-0.851730307,0.431275333],[0,0,0,0],[9E+09,9E+09,9E+09,9E+09,9E+09,9E+09]];
  CONST robtarget Target_1740:=[[-39.710671647,159.052723834,20.366600679],[0.089637387,-0.283764355,-0.851730307,0.431275333],[0,0,0,0],[9E+09,9E+09,9E+09,9E+09,9E+09,9E+09]];
  CONST robtarget Target_1750:=[[-38.675489479,158.720660141,19.88215816],[0.089637387,-0.283764355,-0.851730307,0.431275333],[0,0,0,0],[9E+09,9E+09,9E+09,9E+09,9E+09,9E+09]];
  CONST robtarget Target_1760:=[[-37.650596085,158.370016319,19.404539813],[0.089637387,-0.283764355,-0.851730307,0.431275333],[0,0,0,0],[9E+09,9E+09,9E+09,9E+09,9E+09,9E+09]];
  CONST robtarget Target_1770:=[[-36.636357657,158.001177889,18.933813973],[0.089637387,-0.283764355,-0.851730307,0.431275333],[0,0,0,0],[9E+09,9E+09,9E+09,9E+09,9E+09,9E+09]];
  CONST robtarget Target_1780:=[[-35.633140386,157.614530375,18.470048979],[0.089637387,-0.283764355,-0.851730307,0.431275333],[0,0,0,0],[9E+09,9E+09,9E+09,9E+09,9E+09,9E+09]];
  CONST robtarget Target_1790:=[[-34.641310463,157.210459298,18.013313167],[0.089637387,-0.283764355,-0.851730307,0.431275333],[0,0,0,0],[9E+09,9E+09,9E+09,9E+09,9E+09,9E+09]];
  CONST robtarget Target_1800:=[[-33.661234081,156.789350181,17.563674874],[0.089637387,-0.283764355,-0.851730307,0.431275333],[0,0,0,0],[9E+09,9E+09,9E+09,9E+09,9E+09,9E+09]];
  CONST robtarget Target_1810:=[[-32.69327743,156.351588547,17.121202438],[0.089637387,-0.283764355,-0.851730307,0.431275333],[0,0,0,0],[9E+09,9E+09,9E+09,9E+09,9E+09,9E+09]];
  CONST robtarget Target_1820:=[[-31.737791053,155.897553351,16.685959875],[0.089637387,-0.283764355,-0.851730307,0.431275333],[0,0,0,0],[9E+09,9E+09,9E+09,9E+09,9E+09,9E+09]];
  CONST robtarget Target_1830:=[[-30.795070542,155.427599777,16.257996131],[0.089637387,-0.283764355,-0.851730307,0.431275333],[0,0,0,0],[9E+09,9E+09,9E+09,9E+09,9E+09,9E+09]];
  CONST robtarget Target_1840:=[[-29.865399659,154.942077691,15.837356936],[0.089637387,-0.283764355,-0.851730307,0.431275333],[0,0,0,0],[9E+09,9E+09,9E+09,9E+09,9E+09,9E+09]];
  CONST robtarget Target_1850:=[[-28.949062169,154.44133696,15.424088021],[0.089637387,-0.283764355,-0.851730307,0.431275333],[0,0,0,0],[9E+09,9E+09,9E+09,9E+09,9E+09,9E+09]];
  CONST robtarget Target_1860:=[[-28.046341837,153.92572745,15.018235117],[0.089637387,-0.283764355,-0.851730307,0.431275333],[0,0,0,0],[9E+09,9E+09,9E+09,9E+09,9E+09,9E+09]];
  CONST robtarget Target_1870:=[[-27.157522426,153.395599027,14.619843954],[0.089637387,-0.283764355,-0.851730307,0.431275333],[0,0,0,0],[9E+09,9E+09,9E+09,9E+09,9E+09,9E+09]];
  CONST robtarget Target_1880:=[[-26.2828877,152.851301557,14.228960264],[0.089637387,-0.283764355,-0.851730307,0.431275333],[0,0,0,0],[9E+09,9E+09,9E+09,9E+09,9E+09,9E+09]];
  CONST robtarget Target_1890:=[[-25.422721424,152.293184907,13.845629776],[0.089637387,-0.283764355,-0.851730307,0.431275333],[0,0,0,0],[9E+09,9E+09,9E+09,9E+09,9E+09,9E+09]];
  CONST robtarget Target_1900:=[[-24.577292951,151.721592779,13.469894259],[0.089637387,-0.283764355,-0.851730307,0.431275333],[0,0,0,0],[9E+09,9E+09,9E+09,9E+09,9E+09,9E+09]];
  CONST robtarget Target_1910:=[[-23.746821381,151.136846643,13.101781769],[0.089637387,-0.283764355,-0.851730307,0.431275333],[0,0,0,0],[9E+09,9E+09,9E+09,9E+09,9E+09,9E+09]];
  CONST robtarget Target_1920:=[[-22.931515099,150.539263009,12.741317469],[0.089637387,-0.283764355,-0.851730307,0.431275333],[0,0,0,0],[9E+09,9E+09,9E+09,9E+09,9E+09,9E+09]];
  CONST robtarget Target_1930:=[[-22.131582488,149.929158392,12.388526521],[0.089637387,-0.283764355,-0.851730307,0.431275333],[0,0,0,0],[9E+09,9E+09,9E+09,9E+09,9E+09,9E+09]];
  CONST robtarget Target_1940:=[[-21.347231932,149.306849302,12.043434088],[0.089637387,-0.283764355,-0.851730307,0.431275333],[0,0,0,0],[9E+09,9E+09,9E+09,9E+09,9E+09,9E+09]];
  CONST robtarget Target_1950:=[[-20.578671817,148.672652254,11.706065331],[0.089637387,-0.283764355,-0.851730307,0.431275333],[0,0,0,0],[9E+09,9E+09,9E+09,9E+09,9E+09,9E+09]];
  CONST robtarget Target_1960:=[[-19.826110526,148.026883758,11.376445415],[0.089637387,-0.283764355,-0.851730307,0.431275333],[0,0,0,0],[9E+09,9E+09,9E+09,9E+09,9E+09,9E+09]];
  CONST robtarget Target_1970:=[[-19.089756443,147.369860328,11.0545995],[0.089637387,-0.283764355,-0.851730307,0.431275333],[0,0,0,0],[9E+09,9E+09,9E+09,9E+09,9E+09,9E+09]];
  CONST robtarget Target_1980:=[[-18.369804741,146.701892705,10.740549135],[0.089637387,-0.283764355,-0.851730307,0.431275333],[0,0,0,0],[9E+09,9E+09,9E+09,9E+09,9E+09,9E+09]];
  CONST robtarget Target_1990:=[[-17.666404877,146.023270878,10.434303465],[0.089637387,-0.283764355,-0.851730307,0.431275333],[0,0,0,0],[9E+09,9E+09,9E+09,9E+09,9E+09,9E+09]];
  CONST robtarget Target_2000:=[[-16.979696664,145.334280229,10.135869056],[0.089637387,-0.283764355,-0.851730307,0.431275333],[0,0,0,0],[9E+09,9E+09,9E+09,9E+09,9E+09,9E+09]];
  CONST robtarget Target_2010:=[[-16.309819914,144.635206143,9.845252469],[0.089637387,-0.283764355,-0.851730307,0.431275333],[0,0,0,0],[9E+09,9E+09,9E+09,9E+09,9E+09,9E+09]];
  CONST robtarget Target_2020:=[[-15.656914441,143.926334002,9.562460269],[0.089637387,-0.283764355,-0.851730307,0.431275333],[0,0,0,0],[9E+09,9E+09,9E+09,9E+09,9E+09,9E+09]];
  CONST robtarget Target_2030:=[[-15.021120058,143.207949189,9.287499019],[0.089637387,-0.283764355,-0.851730307,0.431275333],[0,0,0,0],[9E+09,9E+09,9E+09,9E+09,9E+09,9E+09]];
  CONST robtarget Target_2040:=[[-14.402576576,142.480337088,9.020375283],[0.089637387,-0.283764355,-0.851730307,0.431275333],[0,0,0,0],[9E+09,9E+09,9E+09,9E+09,9E+09,9E+09]];
  CONST robtarget Target_2050:=[[-13.801423809,141.743783082,8.761095624],[0.089637387,-0.283764355,-0.851730307,0.431275333],[0,0,0,0],[9E+09,9E+09,9E+09,9E+09,9E+09,9E+09]];
  CONST robtarget Target_2060:=[[-13.217777227,140.998561328,8.509660027],[0.089637387,-0.283764355,-0.851730307,0.431275333],[0,0,0,0],[9E+09,9E+09,9E+09,9E+09,9E+09,9E+09]];
  CONST robtarget Target_2070:=[[-12.651720819,140.244931337,8.266059989],[0.089637387,-0.283764355,-0.851730307,0.431275333],[0,0,0,0],[9E+09,9E+09,9E+09,9E+09,9E+09,9E+09]];
  CONST robtarget Target_2080:=[[-12.103347172,139.483156517,8.030289341],[0.089637387,-0.283764355,-0.851730307,0.431275333],[0,0,0,0],[9E+09,9E+09,9E+09,9E+09,9E+09,9E+09]];
  CONST robtarget Target_2090:=[[-11.572748875,138.713500278,7.802341912],[0.089637387,-0.283764355,-0.851730307,0.431275333],[0,0,0,0],[9E+09,9E+09,9E+09,9E+09,9E+09,9E+09]];
  CONST robtarget Target_2100:=[[-11.060070837,137.936206881,7.582230836],[0.089637387,-0.283764355,-0.851730307,0.431275333],[0,0,0,0],[9E+09,9E+09,9E+09,9E+09,9E+09,9E+09]];
  CONST robtarget Target_2110:=[[-10.565137138,137.151599148,7.369855528],[0.089637387,-0.283764355,-0.851730307,0.431275333],[0,0,0,0],[9E+09,9E+09,9E+09,9E+09,9E+09,9E+09]];
  CONST robtarget Target_2120:=[[-9.626948146,135.561965697,6.967605232],[0.089637387,-0.283764355,-0.851730307,0.431275333],[0,0,0,0],[9E+09,9E+09,9E+09,9E+09,9E+09,9E+09]];
  CONST robtarget Target_2130:=[[-8.754836245,133.947717227,6.594092121],[0.089637387,-0.283764355,-0.851730307,0.431275333],[0,0,0,0],[9E+09,9E+09,9E+09,9E+09,9E+09,9E+09]];
  CONST robtarget Target_2140:=[[-7.945359702,132.311828762,6.247803143],[0.089637387,-0.283764355,-0.851730307,0.431275333],[0,0,0,0],[9E+09,9E+09,9E+09,9E+09,9E+09,9E+09]];
  CONST robtarget Target_2150:=[[-7.195265184,130.657136926,5.927303104],[0.089637387,-0.283764355,-0.851730307,0.431275333],[0,0,0,0],[9E+09,9E+09,9E+09,9E+09,9E+09,9E+09]];
  CONST robtarget Target_2160:=[[-6.501299359,128.986478344,5.631156809],[0.089637387,-0.283764355,-0.851730307,0.431275333],[0,0,0,0],[9E+09,9E+09,9E+09,9E+09,9E+09,9E+09]];
  CONST robtarget Target_2170:=[[-5.860288763,127.302609884,5.357964601],[0.089637387,-0.283764355,-0.851730307,0.431275333],[0,0,0,0],[9E+09,9E+09,9E+09,9E+09,9E+09,9E+09]];
  CONST robtarget Target_2180:=[[-5.269358486,125.607991247,5.106459628],[0.089637387,-0.283764355,-0.851730307,0.431275333],[0,0,0,0],[9E+09,9E+09,9E+09,9E+09,9E+09,9E+09]];
  CONST robtarget Target_2190:=[[-4.725703021,123.905013308,4.875405903],[0.089637387,-0.283764355,-0.851730307,0.431275333],[0,0,0,0],[9E+09,9E+09,9E+09,9E+09,9E+09,9E+09]];
  CONST robtarget Target_2200:=[[-4.226516863,122.196066941,4.66356744],[0.089637387,-0.283764355,-0.851730307,0.431275333],[0,0,0,0],[9E+09,9E+09,9E+09,9E+09,9E+09,9E+09]];
  CONST robtarget Target_2210:=[[-3.769067757,120.483470177,4.469740835],[0.089637387,-0.283764355,-0.851730307,0.431275333],[0,0,0,0],[9E+09,9E+09,9E+09,9E+09,9E+09,9E+09]];
  CONST robtarget Target_2220:=[[-3.350896362,118.769270663,4.292844048],[0.089637387,-0.283764355,-0.851730307,0.431275333],[0,0,0,0],[9E+09,9E+09,9E+09,9E+09,9E+09,9E+09]];
  CONST robtarget Target_2230:=[[-2.969606545,117.055453694,4.131823137],[0.089637387,-0.283764355,-0.851730307,0.431275333],[0,0,0,0],[9E+09,9E+09,9E+09,9E+09,9E+09,9E+09]];
  CONST robtarget Target_2240:=[[-2.622802171,115.344004565,3.985624159],[0.089637387,-0.283764355,-0.851730307,0.431275333],[0,0,0,0],[9E+09,9E+09,9E+09,9E+09,9E+09,9E+09]];
  CONST robtarget Target_2250:=[[-2.308154,113.636842369,3.85322292],[0.089637387,-0.283764355,-0.851730307,0.431275333],[0,0,0,0],[9E+09,9E+09,9E+09,9E+09,9E+09,9E+09]];
  CONST robtarget Target_2260:=[[-2.023581116,111.9356415,3.733705612],[0.089637387,-0.283764355,-0.851730307,0.431275333],[0,0,0,0],[9E+09,9E+09,9E+09,9E+09,9E+09,9E+09]];
  CONST robtarget Target_2270:=[[-1.767059875,110.242020204,3.626183876],[0.089637387,-0.283764355,-0.851730307,0.431275333],[0,0,0,0],[9E+09,9E+09,9E+09,9E+09,9E+09,9E+09]];
  CONST robtarget Target_2280:=[[-1.536566627,108.557596727,3.529769355],[0.089637387,-0.283764355,-0.851730307,0.431275333],[0,0,0,0],[9E+09,9E+09,9E+09,9E+09,9E+09,9E+09]];
  CONST robtarget Target_2290:=[[-1.330138526,106.88392948,3.443600715],[0.089637387,-0.283764355,-0.851730307,0.431275333],[0,0,0,0],[9E+09,9E+09,9E+09,9E+09,9E+09,9E+09]];
  CONST robtarget Target_2300:=[[-1.146037507,105.222356766,3.366916505],[0.089637387,-0.283764355,-0.851730307,0.431275333],[0,0,0,0],[9E+09,9E+09,9E+09,9E+09,9E+09,9E+09]];
  CONST robtarget Target_2310:=[[-0.982577099,103.57416667,3.298978191],[0.089637387,-0.283764355,-0.851730307,0.431275333],[0,0,0,0],[9E+09,9E+09,9E+09,9E+09,9E+09,9E+09]];
  CONST robtarget Target_2320:=[[-0.838070828,101.940647279,3.239047238],[0.089637387,-0.283764355,-0.851730307,0.431275333],[0,0,0,0],[9E+09,9E+09,9E+09,9E+09,9E+09,9E+09]];
  CONST robtarget Target_2330:=[[-0.710887189,100.323032934,3.186409532],[0.089637387,-0.283764355,-0.851730307,0.431275333],[0,0,0,0],[9E+09,9E+09,9E+09,9E+09,9E+09,9E+09]];
  CONST robtarget Target_2340:=[[-0.599596965,98.722361371,3.140440803],[0.089637387,-0.283764355,-0.851730307,0.431275333],[0,0,0,0],[9E+09,9E+09,9E+09,9E+09,9E+09,9E+09]];
  CONST robtarget Target_2350:=[[-0.502817116,97.139625761,3.10053728],[0.089637387,-0.283764355,-0.851730307,0.431275333],[0,0,0,0],[9E+09,9E+09,9E+09,9E+09,9E+09,9E+09]];
  CONST robtarget Target_2360:=[[-0.419164603,95.575819275,3.066095193],[0.089637387,-0.283764355,-0.851730307,0.431275333],[0,0,0,0],[9E+09,9E+09,9E+09,9E+09,9E+09,9E+09]];
  CONST robtarget Target_2370:=[[-0.347305784,94.031887162,3.036532706],[0.089637387,-0.283764355,-0.851730307,0.431275333],[0,0,0,0],[9E+09,9E+09,9E+09,9E+09,9E+09,9E+09]];
  CONST robtarget Target_2380:=[[-0.286087854,92.508600465,3.011348256],[0.089637387,-0.283764355,-0.851730307,0.431275333],[0,0,0,0],[9E+09,9E+09,9E+09,9E+09,9E+09,9E+09]];
  CONST robtarget Target_2390:=[[-0.23439904,91.006691049,2.990058478],[0.089637387,-0.283764355,-0.851730307,0.431275333],[0,0,0,0],[9E+09,9E+09,9E+09,9E+09,9E+09,9E+09]];
  CONST robtarget Target_2400:=[[-0.191127564,89.526890776,2.972180009],[0.089637387,-0.283764355,-0.851730307,0.431275333],[0,0,0,0],[9E+09,9E+09,9E+09,9E+09,9E+09,9E+09]];
  CONST robtarget Target_2410:=[[-0.155200515,88.069901279,2.957246513],[0.089637387,-0.283764355,-0.851730307,0.431275333],[0,0,0,0],[9E+09,9E+09,9E+09,9E+09,9E+09,9E+09]];
  CONST robtarget Target_2420:=[[-0.125712724,86.636254313,2.944866369],[0.089637387,-0.283764355,-0.851730307,0.431275333],[0,0,0,0],[9E+09,9E+09,9E+09,9E+09,9E+09,9E+09]];
  CONST robtarget Target_2430:=[[-0.08261427,83.840896172,2.926280967],[0.089637387,-0.283764355,-0.851730307,0.431275333],[0,0,0,0],[9E+09,9E+09,9E+09,9E+09,9E+09,9E+09]];
  CONST robtarget Target_2440:=[[-0.056032781,81.142526543,2.913966515],[0.089637387,-0.283764355,-0.851730307,0.431275333],[0,0,0,0],[9E+09,9E+09,9E+09,9E+09,9E+09,9E+09]];
  CONST robtarget Target_2450:=[[-0.043048917,78.537720407,2.906816995],[0.089637387,-0.283764355,-0.851730307,0.431275333],[0,0,0,0],[9E+09,9E+09,9E+09,9E+09,9E+09,9E+09]];
  CONST robtarget Target_2460:=[[-0.0411167,76.022616297,2.903894485],[0.089637387,-0.283764355,-0.851730307,0.431275333],[0,0,0,0],[9E+09,9E+09,9E+09,9E+09,9E+09,9E+09]];
  CONST robtarget Target_2470:=[[-0.054549222,72.411596474,2.905814438],[0.089637387,-0.283764355,-0.851730307,0.431275333],[0,0,0,0],[9E+09,9E+09,9E+09,9E+09,9E+09,9E+09]];
  CONST robtarget Target_2480:=[[-0.082166755,68.986528626,2.913297006],[0.089637387,-0.283764355,-0.851730307,0.431275333],[0,0,0,0],[9E+09,9E+09,9E+09,9E+09,9E+09,9E+09]];
  CONST robtarget Target_2490:=[[-0.131718126,64.695350259,2.928466957],[0.089637387,-0.283764355,-0.851730307,0.431275333],[0,0,0,0],[9E+09,9E+09,9E+09,9E+09,9E+09,9E+09]];
  CONST robtarget Target_2500:=[[-0.336493102,50.490109414,2.996479603],[0.089637387,-0.283764355,-0.851730307,0.431275333],[0,0,0,0],[9E+09,9E+09,9E+09,9E+09,9E+09,9E+09]];
  CONST robtarget Target_2510:=[[-0.383691179,46.346372647,3.012638244],[0.089637387,-0.283764355,-0.851730307,0.431275333],[0,0,0,0],[9E+09,9E+09,9E+09,9E+09,9E+09,9E+09]];
  CONST robtarget Target_2520:=[[-0.411149859,42.849734274,3.022078928],[0.089637387,-0.283764355,-0.851730307,0.431275333],[0,0,0,0],[9E+09,9E+09,9E+09,9E+09,9E+09,9E+09]];
  CONST robtarget Target_2530:=[[-0.424693886,39.212854412,3.026737244],[0.089637387,-0.283764355,-0.851730307,0.431275333],[0,0,0,0],[9E+09,9E+09,9E+09,9E+09,9E+09,9E+09]];
  CONST robtarget Target_2540:=[[-0.421044217,36.010335879,3.025410668],[0.089637387,-0.283764355,-0.851730307,0.431275333],[0,0,0,0],[9E+09,9E+09,9E+09,9E+09,9E+09,9E+09]];
  CONST robtarget Target_2550:=[[-0.41907447,35.554875844,3.024714783],[0.089637387,-0.283764355,-0.851730307,0.431275333],[0,0,0,0],[9E+09,9E+09,9E+09,9E+09,9E+09,9E+09]];
  CONST robtarget Target_2560:=[[-0.472314444,35.675387127,3.779323443],[0.089637387,-0.283764355,-0.851730307,0.431275333],[0,0,0,0],[9E+09,9E+09,9E+09,9E+09,9E+09,9E+09]];
  CONST robtarget Target_2570:=[[-0.568581454,35.850375376,4.916493982],[0.089637387,-0.283764355,-0.851730307,0.431275333],[0,0,0,0],[9E+09,9E+09,9E+09,9E+09,9E+09,9E+09]];
  CONST robtarget Target_2580:=[[-0.674745787,36.009651573,5.97035888],[0.089637387,-0.283764355,-0.851730307,0.431275333],[0,0,0,0],[9E+09,9E+09,9E+09,9E+09,9E+09,9E+09]];
  CONST robtarget Target_2590:=[[-0.814413225,36.18238995,7.165708603],[0.089637387,-0.283764355,-0.851730307,0.431275333],[0,0,0,0],[9E+09,9E+09,9E+09,9E+09,9E+09,9E+09]];
  CONST robtarget Target_2600:=[[-0.938637044,36.316036906,8.108570183],[0.089637387,-0.283764355,-0.851730307,0.431275333],[0,0,0,0],[9E+09,9E+09,9E+09,9E+09,9E+09,9E+09]];
  CONST robtarget Target_2610:=[[-1.087512942,36.455290003,9.134680355],[0.089637387,-0.283764355,-0.851730307,0.431275333],[0,0,0,0],[9E+09,9E+09,9E+09,9E+09,9E+09,9E+09]];
  CONST robtarget Target_2620:=[[-1.239353828,36.579195021,10.094804089],[0.089637387,-0.283764355,-0.851730307,0.431275333],[0,0,0,0],[9E+09,9E+09,9E+09,9E+09,9E+09,9E+09]];
  CONST robtarget Target_2630:=[[-1.421822955,36.712085117,11.161645916],[0.089637387,-0.283764355,-0.851730307,0.431275333],[0,0,0,0],[9E+09,9E+09,9E+09,9E+09,9E+09,9E+09]];
  CONST robtarget Target_2640:=[[-1.603081393,36.831650468,12.148657439],[0.089637387,-0.283764355,-0.851730307,0.431275333],[0,0,0,0],[9E+09,9E+09,9E+09,9E+09,9E+09,9E+09]];
  CONST robtarget Target_2650:=[[-1.815892777,36.954857262,13.235289684],[0.089637387,-0.283764355,-0.851730307,0.431275333],[0,0,0,0],[9E+09,9E+09,9E+09,9E+09,9E+09,9E+09]];
  CONST robtarget Target_2660:=[[-2.022814673,37.063195897,14.232044555],[0.089637387,-0.283764355,-0.851730307,0.431275333],[0,0,0,0],[9E+09,9E+09,9E+09,9E+09,9E+09,9E+09]];
  CONST robtarget Target_2670:=[[-2.264008675,37.17571298,15.332867368],[0.089637387,-0.283764355,-0.851730307,0.431275333],[0,0,0,0],[9E+09,9E+09,9E+09,9E+09,9E+09,9E+09]];
  CONST robtarget Target_2680:=[[-2.503019666,37.269792356,16.365865608],[0.089637387,-0.283764355,-0.851730307,0.431275333],[0,0,0,0],[9E+09,9E+09,9E+09,9E+09,9E+09,9E+09]];
  CONST robtarget Target_2690:=[[-2.767711039,37.357437447,17.450227925],[0.089637387,-0.283764355,-0.851730307,0.431275333],[0,0,0,0],[9E+09,9E+09,9E+09,9E+09,9E+09,9E+09]];
  CONST robtarget Target_2700:=[[-3.015538881,37.427824944,18.415711903],[0.089637387,-0.283764355,-0.851730307,0.431275333],[0,0,0,0],[9E+09,9E+09,9E+09,9E+09,9E+09,9E+09]];
  CONST robtarget Target_2710:=[[-3.293975892,37.493926606,19.450770094],[0.089637387,-0.283764355,-0.851730307,0.431275333],[0,0,0,0],[9E+09,9E+09,9E+09,9E+09,9E+09,9E+09]];
  CONST robtarget Target_2720:=[[-3.445545399,37.523997835,19.99475779],[0.089637387,-0.283764355,-0.851730307,0.431275333],[0,0,0,0],[9E+09,9E+09,9E+09,9E+09,9E+09,9E+09]];
  CONST robtarget Target_2730:=[[-3.605818984,37.551372009,20.556577726],[0.089637387,-0.283764355,-0.851730307,0.431275333],[0,0,0,0],[9E+09,9E+09,9E+09,9E+09,9E+09,9E+09]];
  CONST robtarget Target_2740:=[[-3.908296401,37.591217007,21.583102582],[0.089637387,-0.283764355,-0.851730307,0.431275333],[0,0,0,0],[9E+09,9E+09,9E+09,9E+09,9E+09,9E+09]];
  CONST robtarget Target_2750:=[[-4.236986629,37.619005876,22.65445378],[0.089637387,-0.283764355,-0.851730307,0.431275333],[0,0,0,0],[9E+09,9E+09,9E+09,9E+09,9E+09,9E+09]];
  CONST robtarget Target_2760:=[[-4.545606641,37.632275842,23.624158561],[0.089637387,-0.283764355,-0.851730307,0.431275333],[0,0,0,0],[9E+09,9E+09,9E+09,9E+09,9E+09,9E+09]];
  CONST robtarget Target_2770:=[[-4.881147432,37.633259645,24.644107833],[0.089637387,-0.283764355,-0.851730307,0.431275333],[0,0,0,0],[9E+09,9E+09,9E+09,9E+09,9E+09,9E+09]];
  CONST robtarget Target_2780:=[[-5.245016461,37.619462774,25.715007791],[0.089637387,-0.283764355,-0.851730307,0.431275333],[0,0,0,0],[9E+09,9E+09,9E+09,9E+09,9E+09,9E+09]];
  CONST robtarget Target_2790:=[[-5.638661754,37.588391888,26.837602176],[0.089637387,-0.283764355,-0.851730307,0.431275333],[0,0,0,0],[9E+09,9E+09,9E+09,9E+09,9E+09,9E+09]];
  CONST robtarget Target_2800:=[[-6.062970693,37.537743156,28.012491985],[0.089637387,-0.283764355,-0.851730307,0.431275333],[0,0,0,0],[9E+09,9E+09,9E+09,9E+09,9E+09,9E+09]];
  CONST robtarget Target_2810:=[[-6.517267493,37.465672284,29.239736492],[0.089637387,-0.283764355,-0.851730307,0.431275333],[0,0,0,0],[9E+09,9E+09,9E+09,9E+09,9E+09,9E+09]];
  CONST robtarget Target_2820:=[[-6.998161394,37.371132265,30.518485312],[0.089637387,-0.283764355,-0.851730307,0.431275333],[0,0,0,0],[9E+09,9E+09,9E+09,9E+09,9E+09,9E+09]];
  CONST robtarget Target_2830:=[[-7.393199484,37.28236303,31.560418076],[0.089637387,-0.283764355,-0.851730307,0.431275333],[0,0,0,0],[9E+09,9E+09,9E+09,9E+09,9E+09,9E+09]];
  CONST robtarget Target_2840:=[[-7.796288534,37.179620082,32.62159507],[0.089637387,-0.283764355,-0.851730307,0.431275333],[0,0,0,0],[9E+09,9E+09,9E+09,9E+09,9E+09,9E+09]];
  CONST robtarget Target_2850:=[[-8.20610761,37.063247875,33.701409225],[0.089637387,-0.283764355,-0.851730307,0.431275333],[0,0,0,0],[9E+09,9E+09,9E+09,9E+09,9E+09,9E+09]];
  CONST robtarget Target_2860:=[[-8.621335777,36.933590862,34.79925347],[0.089637387,-0.283764355,-0.851730307,0.431275333],[0,0,0,0],[9E+09,9E+09,9E+09,9E+09,9E+09,9E+09]];
  CONST robtarget Target_2870:=[[-9.040898399,36.790922745,35.914542778],[0.089637387,-0.283764355,-0.851730307,0.431275333],[0,0,0,0],[9E+09,9E+09,9E+09,9E+09,9E+09,9E+09]];
  CONST robtarget Target_2880:=[[-9.464090333,36.635366154,37.046755764],[0.089637387,-0.283764355,-0.851730307,0.431275333],[0,0,0,0],[9E+09,9E+09,9E+09,9E+09,9E+09,9E+09]];
  CONST robtarget Target_2890:=[[-9.890192147,36.467001229,38.195395655],[0.089637387,-0.283764355,-0.851730307,0.431275333],[0,0,0,0],[9E+09,9E+09,9E+09,9E+09,9E+09,9E+09]];
  CONST robtarget Target_2900:=[[-10.318626049,36.285780987,39.360011182],[0.089637387,-0.283764355,-0.851730307,0.431275333],[0,0,0,0],[9E+09,9E+09,9E+09,9E+09,9E+09,9E+09]];
  CONST robtarget Target_2910:=[[-11.108271463,35.919299123,41.534631175],[0.089637387,-0.283764355,-0.851730307,0.431275333],[0,0,0,0],[9E+09,9E+09,9E+09,9E+09,9E+09,9E+09]];
  CONST robtarget Target_2920:=[[-11.700490499,35.616784825,43.19094573],[0.089637387,-0.283764355,-0.851730307,0.431275333],[0,0,0,0],[9E+09,9E+09,9E+09,9E+09,9E+09,9E+09]];
  CONST robtarget Target_2930:=[[-11.897795374,35.510997279,43.747747873],[0.089637387,-0.283764355,-0.851730307,0.431275333],[0,0,0,0],[9E+09,9E+09,9E+09,9E+09,9E+09,9E+09]];
  CONST robtarget Target_2940:=[[-12.661310127,35.078889502,45.926428415],[0.089637387,-0.283764355,-0.851730307,0.431275333],[0,0,0,0],[9E+09,9E+09,9E+09,9E+09,9E+09,9E+09]];
  CONST robtarget Target_2950:=[[-13.22369813,34.738939821,47.554692052],[0.089637387,-0.283764355,-0.851730307,0.431275333],[0,0,0,0],[9E+09,9E+09,9E+09,9E+09,9E+09,9E+09]];
  CONST robtarget Target_2960:=[[-13.409335355,34.622895802,48.096323929],[0.089637387,-0.283764355,-0.851730307,0.431275333],[0,0,0,0],[9E+09,9E+09,9E+09,9E+09,9E+09,9E+09]];
  CONST robtarget Target_2970:=[[-14.164751507,34.134501116,50.316760434],[0.089637387,-0.283764355,-0.851730307,0.431275333],[0,0,0,0],[9E+09,9E+09,9E+09,9E+09,9E+09,9E+09]];
  CONST robtarget Target_2980:=[[-14.895403308,33.639567544,52.484292149],[0.089637387,-0.283764355,-0.851730307,0.431275333],[0,0,0,0],[9E+09,9E+09,9E+09,9E+09,9E+09,9E+09]];
  CONST robtarget Target_2990:=[[-15.603404449,33.139125269,54.599827979],[0.089637387,-0.283764355,-0.851730307,0.431275333],[0,0,0,0],[9E+09,9E+09,9E+09,9E+09,9E+09,9E+09]];
  CONST robtarget Target_3000:=[[-16.291584938,32.632083698,56.664559988],[0.089637387,-0.283764355,-0.851730307,0.431275333],[0,0,0,0],[9E+09,9E+09,9E+09,9E+09,9E+09,9E+09]];
  CONST robtarget Target_3010:=[[-17.018667911,32.078049469,58.829591721],[0.089637387,-0.283764355,-0.851730307,0.431275333],[0,0,0,0],[9E+09,9E+09,9E+09,9E+09,9E+09,9E+09]];
  CONST robtarget Target_3020:=[[-17.744292989,31.5070869,60.955253502],[0.089637387,-0.283764355,-0.851730307,0.431275333],[0,0,0,0],[9E+09,9E+09,9E+09,9E+09,9E+09,9E+09]];
  CONST robtarget Target_3030:=[[-18.472931702,30.915026695,63.042520195],[0.089637387,-0.283764355,-0.851730307,0.431275333],[0,0,0,0],[9E+09,9E+09,9E+09,9E+09,9E+09,9E+09]];
  CONST robtarget Target_3040:=[[-18.838902409,30.609710668,64.071754814],[0.089637387,-0.283764355,-0.851730307,0.431275333],[0,0,0,0],[9E+09,9E+09,9E+09,9E+09,9E+09,9E+09]];
  CONST robtarget Target_3050:=[[-19.205813954,30.29725033,65.09098313],[0.089637387,-0.283764355,-0.851730307,0.431275333],[0,0,0,0],[9E+09,9E+09,9E+09,9E+09,9E+09,9E+09]];
  CONST robtarget Target_3060:=[[-19.97512826,29.617397403,67.188955091],[0.089637387,-0.283764355,-0.851730307,0.431275333],[0,0,0,0],[9E+09,9E+09,9E+09,9E+09,9E+09,9E+09]];
  CONST robtarget Target_3070:=[[-20.360381286,29.26220251,68.221360584],[0.089637387,-0.283764355,-0.851730307,0.431275333],[0,0,0,0],[9E+09,9E+09,9E+09,9E+09,9E+09,9E+09]];
  CONST robtarget Target_3080:=[[-20.744338327,28.895776947,69.241801524],[0.089637387,-0.283764355,-0.851730307,0.431275333],[0,0,0,0],[9E+09,9E+09,9E+09,9E+09,9E+09,9E+09]];
  CONST robtarget Target_3090:=[[-21.154366512,28.487955141,70.32622073],[0.089637387,-0.283764355,-0.851730307,0.431275333],[0,0,0,0],[9E+09,9E+09,9E+09,9E+09,9E+09,9E+09]];
  CONST robtarget Target_3100:=[[-21.520036521,28.111611159,71.285936633],[0.089637387,-0.283764355,-0.851730307,0.431275333],[0,0,0,0],[9E+09,9E+09,9E+09,9E+09,9E+09,9E+09]];
  CONST robtarget Target_3110:=[[-21.929736681,27.6817087,72.344335669],[0.089637387,-0.283764355,-0.851730307,0.431275333],[0,0,0,0],[9E+09,9E+09,9E+09,9E+09,9E+09,9E+09]];
  CONST robtarget Target_3120:=[[-22.309539778,27.279666365,73.303790841],[0.089637387,-0.283764355,-0.851730307,0.431275333],[0,0,0,0],[9E+09,9E+09,9E+09,9E+09,9E+09,9E+09]];
  CONST robtarget Target_3130:=[[-22.744934239,26.819531504,74.371887625],[0.089637387,-0.283764355,-0.851730307,0.431275333],[0,0,0,0],[9E+09,9E+09,9E+09,9E+09,9E+09,9E+09]];
  CONST robtarget Target_3140:=[[-23.169596301,26.369769683,75.384679196],[0.089637387,-0.283764355,-0.851730307,0.431275333],[0,0,0,0],[9E+09,9E+09,9E+09,9E+09,9E+09,9E+09]];
  CONST robtarget Target_3150:=[[-23.580092696,25.930815726,76.34212324],[0.089637387,-0.283764355,-0.851730307,0.431275333],[0,0,0,0],[9E+09,9E+09,9E+09,9E+09,9E+09,9E+09]];
  CONST robtarget Target_3160:=[[-23.973327026,25.503693293,77.244247794],[0.089637387,-0.283764355,-0.851730307,0.431275333],[0,0,0,0],[9E+09,9E+09,9E+09,9E+09,9E+09,9E+09]];
  CONST robtarget Target_3170:=[[-24.409616334,25.015146698,78.238519507],[0.089637387,-0.283764355,-0.851730307,0.431275333],[0,0,0,0],[9E+09,9E+09,9E+09,9E+09,9E+09,9E+09]];
  CONST robtarget Target_3180:=[[-24.806661714,24.552319235,79.144801408],[0.089637387,-0.283764355,-0.851730307,0.431275333],[0,0,0,0],[9E+09,9E+09,9E+09,9E+09,9E+09,9E+09]];
  CONST robtarget Target_3190:=[[-25.236824206,24.041083927,80.117597515],[0.089637387,-0.283764355,-0.851730307,0.431275333],[0,0,0,0],[9E+09,9E+09,9E+09,9E+09,9E+09,9E+09]];
  CONST robtarget Target_3200:=[[-25.628692705,23.578552905,80.980541981],[0.089637387,-0.283764355,-0.851730307,0.431275333],[0,0,0,0],[9E+09,9E+09,9E+09,9E+09,9E+09,9E+09]];
  CONST robtarget Target_3210:=[[-25.872608406,23.295941961,81.501586218],[0.089637387,-0.283764355,-0.851730307,0.431275333],[0,0,0,0],[9E+09,9E+09,9E+09,9E+09,9E+09,9E+09]];
  CONST robtarget Target_3220:=[[-26.336430576,22.767606821,82.461156681],[0.089637387,-0.283764355,-0.851730307,0.431275333],[0,0,0,0],[9E+09,9E+09,9E+09,9E+09,9E+09,9E+09]];
  CONST robtarget Target_3230:=[[-26.75908421,22.285804173,83.312730544],[0.089637387,-0.283764355,-0.851730307,0.431275333],[0,0,0,0],[9E+09,9E+09,9E+09,9E+09,9E+09,9E+09]];
  CONST robtarget Target_3240:=[[-27.2647288,21.698850626,84.313864866],[0.089637387,-0.283764355,-0.851730307,0.431275333],[0,0,0,0],[9E+09,9E+09,9E+09,9E+09,9E+09,9E+09]];
  CONST robtarget Target_3250:=[[-27.702454631,21.186772281,85.158169778],[0.089637387,-0.283764355,-0.851730307,0.431275333],[0,0,0,0],[9E+09,9E+09,9E+09,9E+09,9E+09,9E+09]];
  CONST robtarget Target_3260:=[[-28.071793368,20.751310904,85.854657839],[0.089637387,-0.283764355,-0.851730307,0.431275333],[0,0,0,0],[9E+09,9E+09,9E+09,9E+09,9E+09,9E+09]];
  CONST robtarget Target_3270:=[[-28.541923957,20.18803807,86.724083009],[0.089637387,-0.283764355,-0.851730307,0.431275333],[0,0,0,0],[9E+09,9E+09,9E+09,9E+09,9E+09,9E+09]];
  CONST robtarget Target_3280:=[[-28.982897795,19.649749884,87.521188061],[0.089637387,-0.283764355,-0.851730307,0.431275333],[0,0,0,0],[9E+09,9E+09,9E+09,9E+09,9E+09,9E+09]];
  CONST robtarget Target_3290:=[[-29.308528989,19.246881513,88.095224186],[0.089637387,-0.283764355,-0.851730307,0.431275333],[0,0,0,0],[9E+09,9E+09,9E+09,9E+09,9E+09,9E+09]];
  CONST robtarget Target_3300:=[[-29.579108704,18.917792453,88.550574629],[0.089637387,-0.283764355,-0.851730307,0.431275333],[0,0,0,0],[9E+09,9E+09,9E+09,9E+09,9E+09,9E+09]];
  CONST robtarget Target_3310:=[[-31.09799852,19.88463673,88.545493336],[0.089637387,-0.283764355,-0.851730307,0.431275333],[0,0,0,0],[9E+09,9E+09,9E+09,9E+09,9E+09,9E+09]];
  CONST robtarget Target_3320:=[[-32.63262248,20.835589868,88.550232133],[0.089637387,-0.283764355,-0.851730307,0.431275333],[0,0,0,0],[9E+09,9E+09,9E+09,9E+09,9E+09,9E+09]];
  CONST robtarget Target_3330:=[[-35.741789712,22.696349972,88.584940513],[0.089637387,-0.283764355,-0.851730307,0.431275333],[0,0,0,0],[9E+09,9E+09,9E+09,9E+09,9E+09,9E+09]];
  CONST robtarget Target_3340:=[[-38.892044155,24.513127262,88.646240796],[0.089637387,-0.283764355,-0.851730307,0.431275333],[0,0,0,0],[9E+09,9E+09,9E+09,9E+09,9E+09,9E+09]];
  CONST robtarget Target_3350:=[[-42.068819563,26.298976235,88.725674008],[0.089637387,-0.283764355,-0.851730307,0.431275333],[0,0,0,0],[9E+09,9E+09,9E+09,9E+09,9E+09,9E+09]];
  CONST robtarget Target_3360:=[[-61.941679565,-7.890397172,58.129004558],[0.089637387,-0.283764355,-0.851730307,0.431275333],[0,0,0,0],[9E+09,9E+09,9E+09,9E+09,9E+09,9E+09]];
  CONST jointtarget JtHome:=[[0,0,0,0,0,0],[9E+09,9E+09,9E+09,9E+09,9E+09,9E+09]];
  PROC Propeller()
    MoveJ Target_120,v3000,z1,tWeldGun\WObj:=wobjPropeller;
    MoveL Target_130,v300,z1,tWeldGun\WObj:=wobjPropeller;
    MoveL Target_140,v300,z1,tWeldGun\WObj:=wobjPropeller;
    MoveL Target_150,v300,z1,tWeldGun\WObj:=wobjPropeller;
    MoveL Target_160,v300,z1,tWeldGun\WObj:=wobjPropeller;
    MoveL Target_170,v300,z1,tWeldGun\WObj:=wobjPropeller;
    MoveL Target_180,v300,z1,tWeldGun\WObj:=wobjPropeller;
    MoveL Target_190,v300,z1,tWeldGun\WObj:=wobjPropeller;
    MoveL Target_200,v300,z1,tWeldGun\WObj:=wobjPropeller;
    MoveL Target_210,v300,z1,tWeldGun\WObj:=wobjPropeller;
    MoveL Target_220,v300,z1,tWeldGun\WObj:=wobjPropeller;
    MoveL Target_230,v300,z1,tWeldGun\WObj:=wobjPropeller;
    MoveL Target_240,v300,z1,tWeldGun\WObj:=wobjPropeller;
    MoveL Target_250,v300,z1,tWeldGun\WObj:=wobjPropeller;
    MoveL Target_260,v300,z1,tWeldGun\WObj:=wobjPropeller;
    MoveL Target_270,v300,z1,tWeldGun\WObj:=wobjPropeller;
    MoveL Target_280,v300,z1,tWeldGun\WObj:=wobjPropeller;
    MoveL Target_290,v300,z1,tWeldGun\WObj:=wobjPropeller;
    MoveL Target_300,v300,z1,tWeldGun\WObj:=wobjPropeller;
    MoveL Target_310,v300,z1,tWeldGun\WObj:=wobjPropeller;
    MoveL Target_320,v300,z1,tWeldGun\WObj:=wobjPropeller;
    MoveL Target_330,v300,z1,tWeldGun\WObj:=wobjPropeller;
    MoveL Target_340,v300,z1,tWeldGun\WObj:=wobjPropeller;
    MoveL Target_350,v300,z1,tWeldGun\WObj:=wobjPropeller;
    MoveL Target_360,v300,z1,tWeldGun\WObj:=wobjPropeller;
    MoveL Target_370,v300,z1,tWeldGun\WObj:=wobjPropeller;
    MoveL Target_380,v300,z1,tWeldGun\WObj:=wobjPropeller;
    MoveL Target_390,v300,z1,tWeldGun\WObj:=wobjPropeller;
    MoveL Target_400,v300,z1,tWeldGun\WObj:=wobjPropeller;
    MoveL Target_410,v300,z1,tWeldGun\WObj:=wobjPropeller;
    MoveL Target_420,v300,z1,tWeldGun\WObj:=wobjPropeller;
    MoveL Target_430,v300,z1,tWeldGun\WObj:=wobjPropeller;
    MoveL Target_440,v300,z1,tWeldGun\WObj:=wobjPropeller;
    MoveL Target_450,v300,z1,tWeldGun\WObj:=wobjPropeller;
    MoveL Target_460,v300,z1,tWeldGun\WObj:=wobjPropeller;
    MoveL Target_470,v300,z1,tWeldGun\WObj:=wobjPropeller;
    MoveL Target_480,v300,z1,tWeldGun\WObj:=wobjPropeller;
    MoveL Target_490,v300,z1,tWeldGun\WObj:=wobjPropeller;
    MoveL Target_500,v300,z1,tWeldGun\WObj:=wobjPropeller;
    MoveL Target_510,v300,z1,tWeldGun\WObj:=wobjPropeller;
    MoveL Target_520,v300,z1,tWeldGun\WObj:=wobjPropeller;
    MoveL Target_530,v300,z1,tWeldGun\WObj:=wobjPropeller;
    MoveL Target_540,v300,z1,tWeldGun\WObj:=wobjPropeller;
    MoveL Target_550,v300,z1,tWeldGun\WObj:=wobjPropeller;
    MoveL Target_560,v300,z1,tWeldGun\WObj:=wobjPropeller;
    MoveL Target_570,v300,z1,tWeldGun\WObj:=wobjPropeller;
    MoveL Target_580,v300,z1,tWeldGun\WObj:=wobjPropeller;
    MoveL Target_590,v300,z1,tWeldGun\WObj:=wobjPropeller;
    MoveL Target_600,v300,z1,tWeldGun\WObj:=wobjPropeller;
    MoveL Target_610,v300,z1,tWeldGun\WObj:=wobjPropeller;
    MoveL Target_620,v300,z1,tWeldGun\WObj:=wobjPropeller;
    MoveL Target_630,v300,z1,tWeldGun\WObj:=wobjPropeller;
    MoveL Target_640,v300,z1,tWeldGun\WObj:=wobjPropeller;
    MoveL Target_650,v300,z1,tWeldGun\WObj:=wobjPropeller;
    MoveL Target_660,v300,z1,tWeldGun\WObj:=wobjPropeller;
    MoveL Target_670,v300,z1,tWeldGun\WObj:=wobjPropeller;
    MoveL Target_680,v300,z1,tWeldGun\WObj:=wobjPropeller;
    MoveL Target_690,v300,z1,tWeldGun\WObj:=wobjPropeller;
    MoveL Target_700,v300,z1,tWeldGun\WObj:=wobjPropeller;
    MoveL Target_710,v300,z1,tWeldGun\WObj:=wobjPropeller;
    MoveL Target_720,v300,z1,tWeldGun\WObj:=wobjPropeller;
    MoveL Target_730,v300,z1,tWeldGun\WObj:=wobjPropeller;
    MoveL Target_740,v300,z1,tWeldGun\WObj:=wobjPropeller;
    MoveL Target_750,v300,z1,tWeldGun\WObj:=wobjPropeller;
    MoveL Target_760,v300,z1,tWeldGun\WObj:=wobjPropeller;
    MoveL Target_770,v300,z1,tWeldGun\WObj:=wobjPropeller;
    MoveL Target_780,v300,z1,tWeldGun\WObj:=wobjPropeller;
    MoveL Target_790,v300,z1,tWeldGun\WObj:=wobjPropeller;
    MoveL Target_800,v300,z1,tWeldGun\WObj:=wobjPropeller;
    MoveL Target_810,v300,z1,tWeldGun\WObj:=wobjPropeller;
    MoveL Target_820,v300,z1,tWeldGun\WObj:=wobjPropeller;
    MoveL Target_830,v300,z1,tWeldGun\WObj:=wobjPropeller;
    MoveL Target_840,v300,z1,tWeldGun\WObj:=wobjPropeller;
    MoveL Target_850,v300,z1,tWeldGun\WObj:=wobjPropeller;
    MoveL Target_860,v300,z1,tWeldGun\WObj:=wobjPropeller;
    MoveL Target_870,v300,z1,tWeldGun\WObj:=wobjPropeller;
    MoveL Target_880,v300,z1,tWeldGun\WObj:=wobjPropeller;
    MoveL Target_890,v300,z1,tWeldGun\WObj:=wobjPropeller;
    MoveL Target_900,v300,z1,tWeldGun\WObj:=wobjPropeller;
    MoveL Target_910,v300,z1,tWeldGun\WObj:=wobjPropeller;
    MoveL Target_920,v300,z1,tWeldGun\WObj:=wobjPropeller;
    MoveL Target_930,v300,z1,tWeldGun\WObj:=wobjPropeller;
    MoveL Target_940,v300,z1,tWeldGun\WObj:=wobjPropeller;
    MoveL Target_950,v300,z1,tWeldGun\WObj:=wobjPropeller;
    MoveL Target_960,v300,z1,tWeldGun\WObj:=wobjPropeller;
    MoveL Target_970,v300,z1,tWeldGun\WObj:=wobjPropeller;
    MoveL Target_980,v300,z1,tWeldGun\WObj:=wobjPropeller;
    MoveL Target_990,v300,z1,tWeldGun\WObj:=wobjPropeller;
    MoveL Target_1000,v300,z1,tWeldGun\WObj:=wobjPropeller;
    MoveL Target_1010,v300,z1,tWeldGun\WObj:=wobjPropeller;
    MoveL Target_1020,v300,z1,tWeldGun\WObj:=wobjPropeller;
    MoveL Target_1030,v300,z1,tWeldGun\WObj:=wobjPropeller;
    MoveL Target_1040,v300,z1,tWeldGun\WObj:=wobjPropeller;
    MoveL Target_1050,v300,z1,tWeldGun\WObj:=wobjPropeller;
    MoveL Target_1060,v300,z1,tWeldGun\WObj:=wobjPropeller;
    MoveL Target_1070,v300,z1,tWeldGun\WObj:=wobjPropeller;
    MoveL Target_1080,v300,z1,tWeldGun\WObj:=wobjPropeller;
    MoveL Target_1090,v300,z1,tWeldGun\WObj:=wobjPropeller;
    MoveL Target_1100,v300,z1,tWeldGun\WObj:=wobjPropeller;
    MoveL Target_1110,v300,z1,tWeldGun\WObj:=wobjPropeller;
    MoveL Target_1120,v300,z1,tWeldGun\WObj:=wobjPropeller;
    MoveL Target_1130,v300,z1,tWeldGun\WObj:=wobjPropeller;
    MoveL Target_1140,v300,z1,tWeldGun\WObj:=wobjPropeller;
    MoveL Target_1150,v300,z1,tWeldGun\WObj:=wobjPropeller;
    MoveL Target_1160,v300,z1,tWeldGun\WObj:=wobjPropeller;
    MoveL Target_1170,v300,z1,tWeldGun\WObj:=wobjPropeller;
    MoveL Target_1180,v300,z1,tWeldGun\WObj:=wobjPropeller;
    MoveL Target_1190,v300,z1,tWeldGun\WObj:=wobjPropeller;
    MoveL Target_1200,v300,z1,tWeldGun\WObj:=wobjPropeller;
    MoveL Target_1210,v300,z1,tWeldGun\WObj:=wobjPropeller;
    MoveL Target_1220,v300,z1,tWeldGun\WObj:=wobjPropeller;
    MoveL Target_1230,v300,z1,tWeldGun\WObj:=wobjPropeller;
    MoveL Target_1240,v300,z1,tWeldGun\WObj:=wobjPropeller;
    MoveL Target_1250,v300,z1,tWeldGun\WObj:=wobjPropeller;
    MoveL Target_1260,v300,z1,tWeldGun\WObj:=wobjPropeller;
    MoveL Target_1270,v300,z1,tWeldGun\WObj:=wobjPropeller;
    MoveL Target_1280,v300,z1,tWeldGun\WObj:=wobjPropeller;
    MoveL Target_1290,v300,z1,tWeldGun\WObj:=wobjPropeller;
    MoveL Target_1300,v300,z1,tWeldGun\WObj:=wobjPropeller;
    MoveL Target_1310,v300,z1,tWeldGun\WObj:=wobjPropeller;
    MoveL Target_1320,v300,z1,tWeldGun\WObj:=wobjPropeller;
    MoveL Target_1330,v300,z1,tWeldGun\WObj:=wobjPropeller;
    MoveL Target_1340,v300,z1,tWeldGun\WObj:=wobjPropeller;
    MoveL Target_1350,v300,z1,tWeldGun\WObj:=wobjPropeller;
    MoveL Target_1360,v300,z1,tWeldGun\WObj:=wobjPropeller;
    MoveL Target_1370,v300,z1,tWeldGun\WObj:=wobjPropeller;
    MoveL Target_1380,v300,z1,tWeldGun\WObj:=wobjPropeller;
    MoveL Target_1390,v300,z1,tWeldGun\WObj:=wobjPropeller;
    MoveL Target_1400,v300,z1,tWeldGun\WObj:=wobjPropeller;
    MoveL Target_1410,v300,z1,tWeldGun\WObj:=wobjPropeller;
    MoveL Target_1420,v300,z1,tWeldGun\WObj:=wobjPropeller;
    MoveL Target_1430,v300,z1,tWeldGun\WObj:=wobjPropeller;
    MoveL Target_1440,v300,z1,tWeldGun\WObj:=wobjPropeller;
    MoveL Target_1450,v300,z1,tWeldGun\WObj:=wobjPropeller;
    MoveL Target_1460,v300,z1,tWeldGun\WObj:=wobjPropeller;
    MoveL Target_1470,v300,z1,tWeldGun\WObj:=wobjPropeller;
    MoveL Target_1480,v300,z1,tWeldGun\WObj:=wobjPropeller;
    MoveL Target_1490,v300,z1,tWeldGun\WObj:=wobjPropeller;
    MoveL Target_1500,v300,z1,tWeldGun\WObj:=wobjPropeller;
    MoveL Target_1510,v300,z1,tWeldGun\WObj:=wobjPropeller;
    MoveL Target_1520,v300,z1,tWeldGun\WObj:=wobjPropeller;
    MoveL Target_1530,v300,z1,tWeldGun\WObj:=wobjPropeller;
    MoveL Target_1540,v300,z1,tWeldGun\WObj:=wobjPropeller;
    MoveL Target_1550,v300,z1,tWeldGun\WObj:=wobjPropeller;
    MoveL Target_1560,v300,z1,tWeldGun\WObj:=wobjPropeller;
    MoveL Target_1570,v300,z1,tWeldGun\WObj:=wobjPropeller;
    MoveL Target_1580,v300,z1,tWeldGun\WObj:=wobjPropeller;
    MoveL Target_1590,v300,z1,tWeldGun\WObj:=wobjPropeller;
    MoveL Target_1600,v300,z1,tWeldGun\WObj:=wobjPropeller;
    MoveL Target_1610,v300,z1,tWeldGun\WObj:=wobjPropeller;
    MoveL Target_1620,v300,z1,tWeldGun\WObj:=wobjPropeller;
    MoveL Target_1630,v300,z1,tWeldGun\WObj:=wobjPropeller;
    MoveL Target_1640,v300,z1,tWeldGun\WObj:=wobjPropeller;
    MoveL Target_1650,v300,z1,tWeldGun\WObj:=wobjPropeller;
    MoveL Target_1660,v300,z1,tWeldGun\WObj:=wobjPropeller;
    MoveL Target_1670,v300,z1,tWeldGun\WObj:=wobjPropeller;
    MoveL Target_1680,v300,z1,tWeldGun\WObj:=wobjPropeller;
    MoveL Target_1690,v300,z1,tWeldGun\WObj:=wobjPropeller;
    MoveL Target_1700,v300,z1,tWeldGun\WObj:=wobjPropeller;
    MoveL Target_1710,v300,z1,tWeldGun\WObj:=wobjPropeller;
    MoveL Target_1720,v300,z1,tWeldGun\WObj:=wobjPropeller;
    MoveL Target_1730,v300,z1,tWeldGun\WObj:=wobjPropeller;
    MoveL Target_1740,v300,z1,tWeldGun\WObj:=wobjPropeller;
    MoveL Target_1750,v300,z1,tWeldGun\WObj:=wobjPropeller;
    MoveL Target_1760,v300,z1,tWeldGun\WObj:=wobjPropeller;
    MoveL Target_1770,v300,z1,tWeldGun\WObj:=wobjPropeller;
    MoveL Target_1780,v300,z1,tWeldGun\WObj:=wobjPropeller;
    MoveL Target_1790,v300,z1,tWeldGun\WObj:=wobjPropeller;
    MoveL Target_1800,v300,z1,tWeldGun\WObj:=wobjPropeller;
    MoveL Target_1810,v300,z1,tWeldGun\WObj:=wobjPropeller;
    MoveL Target_1820,v300,z1,tWeldGun\WObj:=wobjPropeller;
    MoveL Target_1830,v300,z1,tWeldGun\WObj:=wobjPropeller;
    MoveL Target_1840,v300,z1,tWeldGun\WObj:=wobjPropeller;
    MoveL Target_1850,v300,z1,tWeldGun\WObj:=wobjPropeller;
    MoveL Target_1860,v300,z1,tWeldGun\WObj:=wobjPropeller;
    MoveL Target_1870,v300,z1,tWeldGun\WObj:=wobjPropeller;
    MoveL Target_1880,v300,z1,tWeldGun\WObj:=wobjPropeller;
    MoveL Target_1890,v300,z1,tWeldGun\WObj:=wobjPropeller;
    MoveL Target_1900,v300,z1,tWeldGun\WObj:=wobjPropeller;
    MoveL Target_1910,v300,z1,tWeldGun\WObj:=wobjPropeller;
    MoveL Target_1920,v300,z1,tWeldGun\WObj:=wobjPropeller;
    MoveL Target_1930,v300,z1,tWeldGun\WObj:=wobjPropeller;
    MoveL Target_1940,v300,z1,tWeldGun\WObj:=wobjPropeller;
    MoveL Target_1950,v300,z1,tWeldGun\WObj:=wobjPropeller;
    MoveL Target_1960,v300,z1,tWeldGun\WObj:=wobjPropeller;
    MoveL Target_1970,v300,z1,tWeldGun\WObj:=wobjPropeller;
    MoveL Target_1980,v300,z1,tWeldGun\WObj:=wobjPropeller;
    MoveL Target_1990,v300,z1,tWeldGun\WObj:=wobjPropeller;
    MoveL Target_2000,v300,z1,tWeldGun\WObj:=wobjPropeller;
    MoveL Target_2010,v300,z1,tWeldGun\WObj:=wobjPropeller;
    MoveL Target_2020,v300,z1,tWeldGun\WObj:=wobjPropeller;
    MoveL Target_2030,v300,z1,tWeldGun\WObj:=wobjPropeller;
    MoveL Target_2040,v300,z1,tWeldGun\WObj:=wobjPropeller;
    MoveL Target_2050,v300,z1,tWeldGun\WObj:=wobjPropeller;
    MoveL Target_2060,v300,z1,tWeldGun\WObj:=wobjPropeller;
    MoveL Target_2070,v300,z1,tWeldGun\WObj:=wobjPropeller;
    MoveL Target_2080,v300,z1,tWeldGun\WObj:=wobjPropeller;
    MoveL Target_2090,v300,z1,tWeldGun\WObj:=wobjPropeller;
    MoveL Target_2100,v300,z1,tWeldGun\WObj:=wobjPropeller;
    MoveL Target_2110,v300,z1,tWeldGun\WObj:=wobjPropeller;
    MoveL Target_2120,v300,z1,tWeldGun\WObj:=wobjPropeller;
    MoveL Target_2130,v300,z1,tWeldGun\WObj:=wobjPropeller;
    MoveL Target_2140,v300,z1,tWeldGun\WObj:=wobjPropeller;
    MoveL Target_2150,v300,z1,tWeldGun\WObj:=wobjPropeller;
    MoveL Target_2160,v300,z1,tWeldGun\WObj:=wobjPropeller;
    MoveL Target_2170,v300,z1,tWeldGun\WObj:=wobjPropeller;
    MoveL Target_2180,v300,z1,tWeldGun\WObj:=wobjPropeller;
    MoveL Target_2190,v300,z1,tWeldGun\WObj:=wobjPropeller;
    MoveL Target_2200,v300,z1,tWeldGun\WObj:=wobjPropeller;
    MoveL Target_2210,v300,z1,tWeldGun\WObj:=wobjPropeller;
    MoveL Target_2220,v300,z1,tWeldGun\WObj:=wobjPropeller;
    MoveL Target_2230,v300,z1,tWeldGun\WObj:=wobjPropeller;
    MoveL Target_2240,v300,z1,tWeldGun\WObj:=wobjPropeller;
    MoveL Target_2250,v300,z1,tWeldGun\WObj:=wobjPropeller;
    MoveL Target_2260,v300,z1,tWeldGun\WObj:=wobjPropeller;
    MoveL Target_2270,v300,z1,tWeldGun\WObj:=wobjPropeller;
    MoveL Target_2280,v300,z1,tWeldGun\WObj:=wobjPropeller;
    MoveL Target_2290,v300,z1,tWeldGun\WObj:=wobjPropeller;
    MoveL Target_2300,v300,z1,tWeldGun\WObj:=wobjPropeller;
    MoveL Target_2310,v300,z1,tWeldGun\WObj:=wobjPropeller;
    MoveL Target_2320,v300,z1,tWeldGun\WObj:=wobjPropeller;
    MoveL Target_2330,v300,z1,tWeldGun\WObj:=wobjPropeller;
    MoveL Target_2340,v300,z1,tWeldGun\WObj:=wobjPropeller;
    MoveL Target_2350,v300,z1,tWeldGun\WObj:=wobjPropeller;
    MoveL Target_2360,v300,z1,tWeldGun\WObj:=wobjPropeller;
    MoveL Target_2370,v300,z1,tWeldGun\WObj:=wobjPropeller;
    MoveL Target_2380,v300,z1,tWeldGun\WObj:=wobjPropeller;
    MoveL Target_2390,v300,z1,tWeldGun\WObj:=wobjPropeller;
    MoveL Target_2400,v300,z1,tWeldGun\WObj:=wobjPropeller;
    MoveL Target_2410,v300,z1,tWeldGun\WObj:=wobjPropeller;
    MoveL Target_2420,v300,z1,tWeldGun\WObj:=wobjPropeller;
    MoveL Target_2430,v300,z1,tWeldGun\WObj:=wobjPropeller;
    MoveL Target_2440,v300,z1,tWeldGun\WObj:=wobjPropeller;
    MoveL Target_2450,v300,z1,tWeldGun\WObj:=wobjPropeller;
    MoveL Target_2460,v300,z1,tWeldGun\WObj:=wobjPropeller;
    MoveL Target_2470,v300,z1,tWeldGun\WObj:=wobjPropeller;
    MoveL Target_2480,v300,z1,tWeldGun\WObj:=wobjPropeller;
    MoveL Target_2490,v300,z1,tWeldGun\WObj:=wobjPropeller;
    MoveL Target_2500,v300,z1,tWeldGun\WObj:=wobjPropeller;
    MoveL Target_2510,v300,z1,tWeldGun\WObj:=wobjPropeller;
    MoveL Target_2520,v300,z1,tWeldGun\WObj:=wobjPropeller;
    MoveL Target_2530,v300,z1,tWeldGun\WObj:=wobjPropeller;
    MoveL Target_2540,v300,z1,tWeldGun\WObj:=wobjPropeller;
    MoveL Target_2550,v300,z1,tWeldGun\WObj:=wobjPropeller;
    MoveL Target_2560,v300,z1,tWeldGun\WObj:=wobjPropeller;
    MoveL Target_2570,v300,z1,tWeldGun\WObj:=wobjPropeller;
    MoveL Target_2580,v300,z1,tWeldGun\WObj:=wobjPropeller;
    MoveL Target_2590,v300,z1,tWeldGun\WObj:=wobjPropeller;
    MoveL Target_2600,v300,z1,tWeldGun\WObj:=wobjPropeller;
    MoveL Target_2610,v300,z1,tWeldGun\WObj:=wobjPropeller;
    MoveL Target_2620,v300,z1,tWeldGun\WObj:=wobjPropeller;
    MoveL Target_2630,v300,z1,tWeldGun\WObj:=wobjPropeller;
    MoveL Target_2640,v300,z1,tWeldGun\WObj:=wobjPropeller;
    MoveL Target_2650,v300,z1,tWeldGun\WObj:=wobjPropeller;
    MoveL Target_2660,v300,z1,tWeldGun\WObj:=wobjPropeller;
    MoveL Target_2670,v300,z1,tWeldGun\WObj:=wobjPropeller;
    MoveL Target_2680,v300,z1,tWeldGun\WObj:=wobjPropeller;
    MoveL Target_2690,v300,z1,tWeldGun\WObj:=wobjPropeller;
    MoveL Target_2700,v300,z1,tWeldGun\WObj:=wobjPropeller;
    MoveL Target_2710,v300,z1,tWeldGun\WObj:=wobjPropeller;
    MoveL Target_2720,v300,z1,tWeldGun\WObj:=wobjPropeller;
    MoveL Target_2730,v300,z1,tWeldGun\WObj:=wobjPropeller;
    MoveL Target_2740,v300,z1,tWeldGun\WObj:=wobjPropeller;
    MoveL Target_2750,v300,z1,tWeldGun\WObj:=wobjPropeller;
    MoveL Target_2760,v300,z1,tWeldGun\WObj:=wobjPropeller;
    MoveL Target_2770,v300,z1,tWeldGun\WObj:=wobjPropeller;
    MoveL Target_2780,v300,z1,tWeldGun\WObj:=wobjPropeller;
    MoveL Target_2790,v300,z1,tWeldGun\WObj:=wobjPropeller;
    MoveL Target_2800,v300,z1,tWeldGun\WObj:=wobjPropeller;
    MoveL Target_2810,v300,z1,tWeldGun\WObj:=wobjPropeller;
    MoveL Target_2820,v300,z1,tWeldGun\WObj:=wobjPropeller;
    MoveL Target_2830,v300,z1,tWeldGun\WObj:=wobjPropeller;
    MoveL Target_2840,v300,z1,tWeldGun\WObj:=wobjPropeller;
    MoveL Target_2850,v300,z1,tWeldGun\WObj:=wobjPropeller;
    MoveL Target_2860,v300,z1,tWeldGun\WObj:=wobjPropeller;
    MoveL Target_2870,v300,z1,tWeldGun\WObj:=wobjPropeller;
    MoveL Target_2880,v300,z1,tWeldGun\WObj:=wobjPropeller;
    MoveL Target_2890,v300,z1,tWeldGun\WObj:=wobjPropeller;
    MoveL Target_2900,v300,z1,tWeldGun\WObj:=wobjPropeller;
    MoveL Target_2910,v300,z1,tWeldGun\WObj:=wobjPropeller;
    MoveL Target_2920,v300,z1,tWeldGun\WObj:=wobjPropeller;
    MoveL Target_2930,v300,z1,tWeldGun\WObj:=wobjPropeller;
    MoveL Target_2940,v300,z1,tWeldGun\WObj:=wobjPropeller;
    MoveL Target_2950,v300,z1,tWeldGun\WObj:=wobjPropeller;
    MoveL Target_2960,v300,z1,tWeldGun\WObj:=wobjPropeller;
    MoveL Target_2970,v300,z1,tWeldGun\WObj:=wobjPropeller;
    MoveL Target_2980,v300,z1,tWeldGun\WObj:=wobjPropeller;
    MoveL Target_2990,v300,z1,tWeldGun\WObj:=wobjPropeller;
    MoveL Target_3000,v300,z1,tWeldGun\WObj:=wobjPropeller;
    MoveL Target_3010,v300,z1,tWeldGun\WObj:=wobjPropeller;
    MoveL Target_3020,v300,z1,tWeldGun\WObj:=wobjPropeller;
    MoveL Target_3030,v300,z1,tWeldGun\WObj:=wobjPropeller;
    MoveL Target_3040,v300,z1,tWeldGun\WObj:=wobjPropeller;
    MoveL Target_3050,v300,z1,tWeldGun\WObj:=wobjPropeller;
    MoveL Target_3060,v300,z1,tWeldGun\WObj:=wobjPropeller;
    MoveL Target_3070,v300,z1,tWeldGun\WObj:=wobjPropeller;
    MoveL Target_3080,v300,z1,tWeldGun\WObj:=wobjPropeller;
    MoveL Target_3090,v300,z1,tWeldGun\WObj:=wobjPropeller;
    MoveL Target_3100,v300,z1,tWeldGun\WObj:=wobjPropeller;
    MoveL Target_3110,v300,z1,tWeldGun\WObj:=wobjPropeller;
    MoveL Target_3120,v300,z1,tWeldGun\WObj:=wobjPropeller;
    MoveL Target_3130,v300,z1,tWeldGun\WObj:=wobjPropeller;
    MoveL Target_3140,v300,z1,tWeldGun\WObj:=wobjPropeller;
    MoveL Target_3150,v300,z1,tWeldGun\WObj:=wobjPropeller;
    MoveL Target_3160,v300,z1,tWeldGun\WObj:=wobjPropeller;
    MoveL Target_3170,v300,z1,tWeldGun\WObj:=wobjPropeller;
    MoveL Target_3180,v300,z1,tWeldGun\WObj:=wobjPropeller;
    MoveL Target_3190,v300,z1,tWeldGun\WObj:=wobjPropeller;
    MoveL Target_3200,v300,z1,tWeldGun\WObj:=wobjPropeller;
    MoveL Target_3210,v300,z1,tWeldGun\WObj:=wobjPropeller;
    MoveL Target_3220,v300,z1,tWeldGun\WObj:=wobjPropeller;
    MoveL Target_3230,v300,z1,tWeldGun\WObj:=wobjPropeller;
    MoveL Target_3240,v300,z1,tWeldGun\WObj:=wobjPropeller;
    MoveL Target_3250,v300,z1,tWeldGun\WObj:=wobjPropeller;
    MoveL Target_3260,v300,z1,tWeldGun\WObj:=wobjPropeller;
    MoveL Target_3270,v300,z1,tWeldGun\WObj:=wobjPropeller;
    MoveL Target_3280,v300,z1,tWeldGun\WObj:=wobjPropeller;
    MoveL Target_3290,v300,z1,tWeldGun\WObj:=wobjPropeller;
    MoveL Target_3300,v300,z1,tWeldGun\WObj:=wobjPropeller;
    MoveL Target_3310,v300,z1,tWeldGun\WObj:=wobjPropeller;
    MoveL Target_3320,v300,z1,tWeldGun\WObj:=wobjPropeller;
    MoveL Target_3330,v300,z1,tWeldGun\WObj:=wobjPropeller;
    MoveL Target_3340,v300,z1,tWeldGun\WObj:=wobjPropeller;
    MoveL Target_3350,v300,z1,tWeldGun\WObj:=wobjPropeller;
    MoveL Target_3360,v300,z1,tWeldGun\WObj:=wobjPropeller;
  ENDPROC
  PROC Main()
    MoveAbsJ JtHome,v1000,z100,tWeldGun\WObj:=wobjPropeller;
    Propeller;
    MoveAbsJ JtHome,v1000,z100,tWeldGun\WObj:=wobjPropeller;
  ENDPROC
ENDMODULE

